Yaskawa INFORM job: X2_8B-21B(90,180).JBI

/JOB
//NAME X2_8B-21B(90,180)
///FOLDERNAME X2
//POS
///NPOS 931,931,931,42,0,0
///TOOL 0
///POSTYPE PULSE
///PULSE
C00000=-1415,-134459,-133802,-1969,12985,79332
C00001=-87080,-112473,-103627,-41798,51237,70410
C00002=-91681,-107347,-99471,-39221,49165,68848
C00003=-93439,-105106,-97054,-38371,48113,68361
C00004=-93441,-104864,-95967,-38672,47682,68565
C00005=-93504,-104969,-96260,-38564,47753,68495
C00006=-95585,-102642,-95415,-36914,47385,67494
C00007=-93504,-104969,-96260,-38564,47753,68495
C00008=-87147,-112175,-102116,-42180,50619,70689
C00009=-87145,-119394,-106475,-25944,48524,38750
C00010=-91166,-110510,-101811,-22693,48895,36705
C00011=-92650,-107060,-99920,-21494,49065,35962
C00012=-94767,-104655,-99060,-19829,49198,34943
C00013=-94484,-105085,-99259,-20052,49173,35080
C00014=-93721,-102513,-96995,-20598,49294,35408
C00015=-94484,-105085,-99259,-20052,49173,35080
C00016=-89209,-117497,-105909,-24366,48468,37757
C00017=-93166,-113214,-115710,-1969,57926,79332
C00018=-93710,-106990,-108704,-1652,56802,79139
C00019=-93766,-106412,-107148,-1629,56140,79127
C00020=-93768,-106433,-106329,-1638,55626,79135
C00021=-93918,-105383,-106173,-1535,56065,79069
C00022=-94164,-101296,-104676,-1361,57240,78956
C00023=-93895,-105502,-106499,-1547,56205,79076
C00024=-93151,-113316,-114305,-1998,57010,79354
C00025=-81072,-99391,-111155,-4750,63110,78553
C00026=-81984,-95120,-104767,-4287,61328,78293
C00027=-82103,-94682,-103397,-4241,60705,78273
C00028=-82106,-94924,-102383,-4271,59960,78300
C00029=-82089,-94934,-102578,-4276,60076,78302
C00030=-82803,-90374,-100753,-3806,61258,77993
C00031=-82089,-94934,-102578,-4276,60076,78302
C00032=-81057,-100006,-109908,-4804,62030,78604
C00033=-94004,-119945,-107122,49530,42714,48164
C00034=-93972,-116281,-97047,53343,39935,45878
C00035=-92833,-103149,-88492,51302,40218,47068
C00036=-93174,-100930,-87132,51219,40604,47120
C00037=-93174,-100493,-85792,51770,40220,46795
C00038=-93174,-101015,-87399,51095,40684,47186
C00039=-92955,-97894,-86230,50180,41136,47726
C00040=-93303,-100448,-87190,51023,40860,47230
C00041=-98055,-98607,-86499,53149,43882,46024
C00042=-96642,-96320,-85623,51883,43475,46780
C00043=-95342,-96864,-85830,51299,42647,47109
C00044=-97130,-98187,-86063,52744,43317,46271
C00045=-114545,-105110,-100746,39625,57097,48369
C00046=-113947,-102413,-97570,39574,56382,48359
C00047=-113947,-102278,-96691,39772,56015,48196
C00048=-113346,-99976,-96570,39024,56612,48763
C00049=-112899,-98120,-95866,38597,56823,49078
C00050=-114020,-99555,-96940,39169,57262,48705
C00051=-56302,-84822,-83054,-58022,66572,84014
C00052=-58361,-85953,-83540,-57558,65172,83717
C00053=-56302,-84822,-83054,-58022,66572,84014
C00054=-50122,-85714,-86741,-59061,71306,84454
C00055=-54195,-101901,-111197,-24063,62262,77343
C00056=-67243,-111926,-101536,21450,29925,69540
C00057=-66442,-101704,-94400,19916,30532,70304
C00058=-66308,-99858,-92576,19846,30336,70336
C00059=-66311,-99589,-91307,20230,29731,70137
C00060=-66308,-99960,-93112,19687,30597,70418
C00061=-70591,-100617,-92786,25268,31264,67678
C00062=-70591,-100325,-91437,25755,30647,67424
C00063=-68222,-99738,-91214,22742,30105,68906
C00064=-70591,-100606,-92729,25289,31242,67667
C00065=-66097,-110297,-96199,21577,27345,69446
C00066=-65719,-107666,-92844,21562,26575,69447
C00067=-65848,-106528,-92445,21497,26927,69482
C00068=-65365,-110699,-93884,21743,25627,69354
C00069=-67243,-111926,-101536,21450,29925,69540
C00070=-68963,-41843,-96211,-398,96948,-48811
C00071=-76932,-51697,-92360,2602,89609,-51106
C00072=-71886,-45093,-85416,705,88639,-49643
C00073=-71886,-45937,-84760,705,87803,-49648
C00074=-71886,-44632,-85753,705,89084,-49641
C00075=-68776,-90352,-95136,-4313,51281,-47645
C00076=-68803,-86754,-93636,-4241,52203,-47695
C00077=-68762,-92243,-95906,-4353,50785,-47617
C00078=-77446,-64871,-91176,8832,74282,-49527
C00079=-75907,-64612,-91046,8095,74185,-49034
C00080=-78150,-64967,-91224,9168,74335,-49752
C00081=-78150,-57569,-97635,8943,81990,-49191
C00082=-68963,-41843,-96211,-398,96948,-48811
C00083=-67385,-42511,-92598,-992,94393,-48367
C00084=-66773,-44328,-90253,-1220,92024,-48175
C00085=-66900,-44765,-89647,-1171,91425,-48205
C00086=-66773,-43962,-90441,-1221,92327,-48178
C00087=-69817,-49291,-93527,-72,91467,-49038
C00088=-102407,-61387,-79216,48101,75803,-74984
C00089=-99741,-62884,-79905,47237,74215,-74494
C00090=-102407,-61387,-79216,48101,75803,-74984
C00091=-71396,-101707,-96198,105,39560,-49678
C00092=-71544,-99303,-95354,247,40276,-49753
C00093=-71126,-105930,-97636,-165,38275,-49535
C00094=-74447,-120283,-111838,3099,39699,-51260
C00095=-57750,-84762,-113304,-22338,79933,-80646
C00096=-38298,-117376,-123136,-35520,84192,-83183
C00097=-31003,-114098,-105660,-45955,85390,-81321
C00098=-32496,-116782,-107403,-45795,84408,-81579
C00099=-34116,-118987,-108120,-45640,83088,-81742
C00100=-33779,-118873,-108083,-45678,83285,-81673
C00101=-33779,-118389,-106291,-45736,82677,-81394
C00102=-33116,-116007,-107005,-45711,84199,-81779
C00103=-43122,-77390,-91933,-43525,86904,-87571
C00104=-44353,-78017,-92219,-43231,86215,-87819
C00105=-45440,-79271,-92786,-42975,85486,-87990
C00106=-45102,-79332,-92813,-43057,85636,-87902
C00107=-45102,-79709,-91490,-43095,84888,-87585
C00108=-41853,-68825,-87871,-43817,88900,-87868
C00109=-48095,-31712,-66541,-47290,99218,-86920
C00110=-48762,-33638,-67810,-47108,98755,-86994
C00111=-49503,-35735,-69173,-46902,98237,-87073
C00112=-49389,-35416,-68966,-46933,98317,-87062
C00113=-49389,-36060,-68028,-46814,97684,-86756
C00114=-48487,-32850,-67294,-47182,98948,-86964
C00115=-45126,-25671,-76382,-49967,106798,-89554
C00116=-48508,-32956,-85951,-38791,109748,-85822
C00117=-73491,-115415,-129730,-12591,84406,-82629
C00118=-68604,-111632,-124361,34026,103601,-55041
C00119=-52690,-105642,-114364,31889,95098,-51390
C00120=-51347,-103959,-112740,31690,94497,-51045
C00121=-51347,-104280,-111882,31650,93903,-51212
C00122=-50963,-109237,-114816,31559,93129,-51281
C00123=-54701,-101748,-112541,32228,96580,-51739
C00124=-54580,-102143,-110625,32107,95358,-52042
C00125=-52710,-105778,-111943,31798,93771,-51772
C00126=-54580,-102143,-110625,32107,95358,-52042
C00127=-53574,-106836,-112314,31893,93817,-52092
C00128=-52008,-102475,-110737,31756,94333,-51344
C00129=-53574,-106836,-112314,31893,93817,-52092
C00130=-61074,-96775,-114868,33501,102293,-52496
C00131=-149084,-102156,-129577,22032,95315,-42360
C00132=-128569,-114069,-129208,14930,94899,-36248
C00133=-124702,-111484,-125119,14131,93099,-35189
C00134=-123206,-111006,-122572,13804,91571,-34868
C00135=-123205,-111346,-122108,13798,91123,-34918
C00136=-123169,-110975,-122344,13795,91444,-34870
C00137=-122647,-104244,-120003,13724,93323,-34489
C00138=-123169,-110975,-122344,13795,91444,-34870
C00139=-116503,-109521,-121739,12400,90787,-32743
C00140=-113941,-110266,-121994,11839,90202,-31960
C00141=-116503,-109521,-121739,12400,90787,-32743
C00142=-121595,-114825,-128025,13496,92670,-34216
C00143=-123984,-121300,-124584,22039,85383,-28695
C00144=-118596,-113071,-118409,20758,84424,-26972
C00145=-117828,-112575,-117002,20585,83663,-26833
C00146=-117596,-112721,-116348,20543,83158,-26838
C00147=-117643,-112201,-116474,20543,83493,-26797
C00148=-117846,-106122,-114344,20549,85245,-26570
C00149=-117643,-112201,-116474,20543,83493,-26797
C00150=-125192,-113488,-115877,22341,84450,-29296
C00151=-124919,-116220,-115928,22323,83104,-29449
C00152=-122352,-116155,-116251,21738,82647,-28614
C00153=-124919,-116220,-115928,22323,83104,-29449
C00154=-123984,-121300,-124584,22039,85383,-28695
C00155=-86442,-134681,-133724,-19248,79211,-32552
C00156=-86002,-121949,-124889,-19319,80358,-32581
C00157=-85994,-121959,-123892,-19351,79775,-32484
C00158=-85995,-122137,-123177,-19379,79272,-32404
C00159=-85938,-122450,-123568,-19392,79360,-32398
C00160=-86651,-115539,-121342,-19081,81262,-32951
C00161=-85938,-122450,-123568,-19392,79360,-32398
C00162=-130270,-119263,-121891,15868,79169,-48216
C00163=-132135,-133974,-122544,16883,72658,-49767
C00164=-129371,-136174,-123179,16117,71390,-48932
C00165=-132135,-133974,-122544,16883,72658,-49767
C00166=-120611,-122953,-119681,21560,80854,-22535
C00167=-120610,-122943,-118608,21593,80243,-22645
C00168=-120610,-122853,-116921,21650,79318,-22813
C00169=-120610,-122881,-117271,21638,79506,-22779
C00170=-120610,-122878,-117279,21638,79511,-22778
C00171=-120610,-122881,-117271,21638,79506,-22779
C00172=-120610,-122873,-117198,21640,79468,-22785
C00173=-120610,-122853,-117190,21640,79473,-22785
C00174=-120610,-122873,-117198,21640,79468,-22785
C00175=-120611,-122910,-120952,21522,81605,-22399
C00176=-120612,-120891,-127143,3106,87300,-4415
C00177=-120611,-122177,-124352,3111,84925,-4474
C00178=-120611,-122645,-122467,3116,83527,-4507
C00179=-120611,-122779,-121606,3119,82929,-4523
C00180=-120611,-122697,-122159,3117,83311,-4513
C00181=-120611,-122692,-122166,3117,83318,-4513
C00182=-120611,-122697,-122159,3117,83311,-4513
C00183=-120611,-121412,-126223,3107,86468,-4436
C00184=-96873,-136971,-131305,19961,95014,-27830
C00185=-53188,-122774,-119059,34227,101931,-42117
C00186=-53187,-122644,-116623,34032,100735,-42492
C00187=-53184,-122447,-115007,33919,99986,-42724
C00188=-53180,-122268,-113886,33849,99484,-42877
C00189=-53186,-122531,-115629,33961,100272,-42636
C00190=-53233,-122033,-113114,32057,113501,-44659
C00191=-53229,-122037,-113108,32057,113495,-44659
C00192=-53233,-122033,-113114,32057,113501,-44659
C00193=-53127,-122157,-112856,34567,84618,-41563
C00194=-53132,-122146,-112848,34568,84621,-41564
C00195=-53127,-122157,-112856,34567,84618,-41563
C00196=-53124,-122720,-116247,34514,86111,-41098
C00197=-68676,-133744,-131015,10578,108811,-68614
C00198=-80160,-118182,-130261,-41,125141,-81817
C00199=-80187,-122370,-123619,-70,118933,-81856
C00200=-80183,-122639,-122398,-68,118043,-81854
C00201=-80181,-122756,-121636,-67,117515,-81853
C00202=-80184,-122603,-122588,-68,118179,-81854
C00203=-80182,-122615,-122584,-67,118170,-81853
C00204=-80184,-122603,-122588,-68,118179,-81854
C00205=-80200,-121154,-126606,-75,121396,-81862
C00206=-109164,-117358,-132635,-7350,119146,-48306
C00207=-144183,-119511,-130571,-15498,107286,-7245
C00208=-197934,-122815,-127402,-28006,89082,55776
C00209=-202772,-123889,-124791,-27048,85608,54814
C00210=-204705,-124106,-122314,-26692,83530,54575
C00211=-204705,-124189,-120905,-26732,82711,54762
C00212=-205113,-122699,-120601,-26621,83104,54520
C00213=-208506,-122040,-120392,-25870,82241,53457
C00214=-204510,-125657,-121990,-26775,82699,54838
C00215=-204510,-125393,-124777,-26704,84359,54459
C00216=-217123,-144581,-130617,-26990,80795,43719
C00217=-208514,-157553,-136215,-22784,79668,13108
C00218=-208514,-151468,-127497,-22936,77598,13510
C00219=-209226,-147410,-126429,-22728,78719,13024
C00220=-208514,-151468,-127497,-22936,77598,13510
C00221=-208514,-156517,-134755,-22805,79329,13174
C00222=-187736,-116553,-120968,-36188,98329,31010
C00223=-144869,-104708,-130913,697,92502,-12445
C00224=-97478,-100538,-119508,25976,122096,-72949
C00225=-94415,-115583,-120723,24602,114867,-73486
C00226=-94145,-116737,-119872,24403,113768,-73630
C00227=-94090,-116915,-118863,24267,113100,-73760
C00228=-94227,-118887,-121662,24392,113788,-73658
C00229=-94618,-126072,-123928,23885,111795,-74261
C00230=-93811,-121058,-122280,24303,112998,-73673
C00231=-123165,-134656,-120887,30393,109989,-65140
C00232=-122877,-135920,-118822,30065,108215,-65520
C00233=-120918,-135771,-118381,30417,107339,-64954
C00234=-122877,-135920,-118822,30065,108215,-65520
C00235=-123434,-129548,-123417,31323,113703,-64157
C00236=-126606,-101457,-128935,16844,101795,-36174
C00237=-152779,-135138,-131563,2515,76140,-19155
C00238=-150820,-122490,-124749,1875,78392,-18455
C00239=-150097,-118368,-121531,1645,78513,-18212
C00240=-150095,-118599,-120646,1648,77850,-18220
C00241=-147666,-112236,-119185,871,80184,-17389
C00242=-146670,-110099,-118456,556,80825,-17059
C00243=-148658,-114325,-119887,1186,79554,-17722
C00244=-87079,-91764,-103818,-42328,107533,9448
C00245=-87027,-91004,-101788,-42122,106912,9740
C00246=-89264,-90509,-101588,-42089,105978,9119
C00247=-87027,-91004,-101788,-42122,106912,9740
C00248=-87391,-90282,-107909,-43186,109836,8282
C00249=-92115,-87061,-118989,-19004,94950,-3823
C00250=-78975,-130870,-123203,19746,71053,-12291
C00251=-74317,-97013,-111518,17407,83606,-9286
C00252=-74211,-95430,-110119,17377,83539,-9259
C00253=-74211,-95892,-109317,17397,82840,-9358
C00254=-75305,-113551,-114600,17838,69768,-10493
C00255=-78326,-111051,-111958,19079,70114,-11550
C00256=-78379,-106110,-110225,18937,71523,-11339
C00257=-78263,-116865,-113913,19272,68408,-11810
C00258=-85880,-113569,-112821,22054,71256,-14152
C00259=-85920,-114580,-110580,22309,69503,-14507
C00260=-82054,-114988,-110714,20879,68380,-13249
C00261=-85920,-114580,-110580,22309,69503,-14507
C00262=-78975,-130870,-123203,19746,67177,-12291
C00263=-159950,-115131,-126913,-23322,109234,64770
C00264=-163413,-124246,-126581,-22686,103792,64589
C00265=-164859,-127477,-125491,-22457,101245,64551
C00266=-164857,-127553,-124648,-22406,100728,64651
C00267=-164862,-127370,-126252,-22506,101730,64457
C00268=-158275,-145382,-129341,-21795,96649,67831
C00269=-159759,-153222,-131425,-21726,93697,67826
C00270=-158275,-145382,-129341,-21795,96649,67831
C00271=-157577,-144643,-126617,-21696,95625,68274
C00272=-160219,-140867,-125578,-21868,96138,67212
C00273=-157577,-144643,-126617,-21696,95625,68274
C00274=-152631,-134238,-128202,-21932,102817,68768
C00275=-146941,-123801,-133763,-3444,102850,52685
C00276=-136178,-116173,-124987,31736,84906,22811
C00277=-134413,-106132,-117362,31242,84680,23412
C00278=-134231,-105594,-115694,31219,83968,23286
C00279=-134230,-105863,-115134,31239,83552,23172
C00280=-134007,-104199,-114803,31151,84035,23389
C00281=-133473,-100630,-113499,30965,84737,23780
C00282=-134315,-106237,-115533,31260,83629,23161
C00283=-136272,-117460,-124003,31807,83855,22481
C00284=-136226,-116324,-125056,31750,84893,22789
C00285=-134474,-106353,-117504,31259,84679,23389
C00286=-134275,-105758,-115681,31235,83904,23252
C00287=-134274,-105987,-115198,31252,83547,23154
C00288=-134027,-104733,-115029,31162,83924,23350
C00289=-133465,-100971,-113658,30966,84667,23763
C00290=-134308,-106598,-115693,31262,83551,23142
C00291=-136269,-117902,-124178,31812,83752,22453
C00292=-139753,-124875,-130430,383,75663,-26245
C00293=-143223,-157944,-133481,-5653,58679,-38405
C00294=-140983,-144085,-126452,-6488,61628,-37698
C00295=-140148,-138933,-122655,-6835,62006,-37402
C00296=-140147,-138616,-121921,-6853,61719,-37384
C00297=-140691,-136506,-121897,-6553,62737,-37651
C00298=-138669,-131542,-120459,-7325,64564,-37004
C00299=-140691,-136506,-121897,-6553,62737,-37651
C00300=-145148,-139028,-124584,-4588,62787,-39337
C00301=-159973,-92454,-110285,14523,90938,-48717
C00302=-158765,-97223,-112137,14224,89465,-48492
C00303=-159973,-92454,-110285,14523,90938,-48717
C00304=-164681,-91509,-114703,15696,94847,-49769
C00305=-142525,-105883,-132766,-7713,103357,-60336
C00306=-90751,-115691,-121566,-36045,104861,-61043
C00307=-92920,-122587,-117773,-35137,99152,-60047
C00308=-93124,-123070,-117553,-35091,98753,-60003
C00309=-93124,-123008,-116878,-35050,98435,-59900
C00310=-93160,-123063,-117190,-35068,98555,-59953
C00311=-95752,-125144,-117838,-34977,96947,-60505
C00312=-93160,-123063,-117190,-35068,98555,-59953
C00313=-92038,-109836,-114685,-38536,89453,-57060
C00314=-86810,-100893,-104585,-47463,92019,-56975
C00315=-88449,-102594,-103600,-47188,90148,-56855
C00316=-88449,-102618,-102426,-47172,89639,-56610
C00317=-88449,-102603,-103366,-47184,90046,-56806
C00318=-85133,-99388,-102162,-47637,92393,-56350
C00319=-85168,-99488,-101153,-47595,91912,-56132
C00320=-86978,-101259,-101820,-47360,90627,-56378
C00321=-84037,-98201,-102123,-47804,93363,-56297
C00322=-108771,-112096,-123986,-16313,85813,-59347
C00323=-109769,-112695,-132242,-3132,99947,-61138
C00324=-127404,-127157,-120795,27540,73197,-60883
C00325=-120526,-123085,-115007,25540,69700,-59025
C00326=-119461,-122312,-114032,25210,69192,-58723
C00327=-119461,-122116,-113003,25293,68708,-58832
C00328=-119461,-122312,-114032,25210,69192,-58723
C00329=-94655,-112249,-115827,-1041,75214,-51009
C00330=-93364,-111129,-115444,-1499,75574,-50577
C00331=-121213,-123445,-114215,25873,69302,-59387
C00332=-127714,-127278,-119628,27738,72603,-61150
C00333=-140848,-129628,-128054,17424,84805,-27418
C00334=-127903,-106251,-120637,17388,91568,-15860
C00335=-124887,-98361,-114445,16717,91208,-14907
C00336=-124614,-94849,-112077,16660,91489,-14780
C00337=-117832,-103976,-115449,15062,87719,-13014
C00338=-118209,-109888,-118953,15141,86934,-13233
C00339=-120968,-118649,-124805,15800,86569,-14208
C00340=-112726,-101228,-128594,1890,90279,15897
C00341=-102865,-105549,-130121,-1361,88970,18873
C00342=-85416,-143080,-122146,-23399,58401,32529
C00343=-89847,-131888,-116792,-20882,59491,30436
C00344=-92125,-126361,-114096,-19602,60042,29398
C00345=-92108,-126361,-114086,-19611,60041,29405
C00346=-94963,-119193,-112807,-13876,65309,25883
C00347=-99230,-109273,-111594,-7832,72910,21884
C00348=-97558,-114678,-114533,-8498,72116,22521
C00349=-94805,-124749,-120489,-9597,70928,23580
C00350=-89899,-115674,-129227,-15589,81503,27304
C00351=-94000,-113154,-130859,1035,116659,-75004
C00352=-93721,-118000,-129934,5060,122177,-74127
C00353=-93715,-120352,-127357,4900,119392,-74256
C00354=-95346,-120435,-125547,4467,118331,-74923
C00355=-87734,-123112,-126247,6115,116903,-72103
C00356=-93725,-120284,-127319,4898,119404,-74259
C00357=-93731,-117931,-129895,5059,122189,-74130
C00358=-92605,-107385,-114202,-42080,118626,-78084
C00359=-94957,-117308,-114744,-40643,113912,-77125
C00360=-96859,-119647,-113709,-40343,111617,-77062
C00361=-96820,-119688,-113698,-40330,111613,-77042
C00362=-92369,-120637,-111842,-39132,112371,-75247
C00363=-87506,-133441,-114197,-38673,106213,-75021
C00364=-90618,-118755,-112828,-39302,114392,-75239
C00365=-88476,-109244,-112462,-40625,118981,-76164
C00366=-73726,-95231,-122050,-23824,117115,-78775
C00367=-68964,-113071,-130294,19412,109419,-80322
C00368=-55630,-112625,-122011,35520,97927,-81697
C00369=-52390,-118820,-120628,34805,93310,-81881
C00370=-47869,-106069,-116317,31727,98681,-78960
C00371=-58944,-112669,-113031,37596,97582,-82877
C00372=-56690,-122472,-119439,35129,92879,-83747
C00373=-59872,-116629,-120975,35716,97415,-83571
C00374=-61517,-148095,-119735,48293,75564,-80066
C00375=-55473,-148057,-116974,48060,71191,-79214
C00376=-53771,-146175,-114985,47935,70110,-78894
C00377=-54494,-144748,-112549,48210,69974,-79344
C00378=-55476,-147094,-115701,48129,70996,-79318
C00379=-61520,-147186,-118480,48348,75358,-80173
C00380=-69196,-132761,-125763,48066,87564,-77891
C00381=-67178,-112107,-133350,-9560,121946,-71499
C00382=-53652,-115588,-130730,-10921,119132,-80041
C00383=-53631,-118653,-128170,-10572,116038,-79726
C00384=-49406,-129162,-130962,-9295,109096,-77614
C00385=-56866,-119557,-126808,-10903,114346,-80761
C00386=-54665,-117852,-125979,-10629,114989,-80007
C00387=-57520,-119011,-127190,-3009,114777,-80027
C00388=-59278,-121853,-127991,842,113579,-80159
C00389=-55695,-120300,-124998,1328,112531,-78914
C00390=-53493,-120154,-126714,1639,113579,-78070
C00391=-53512,-117734,-129516,1682,116546,-78033
C00392=-64263,-112177,-127274,18013,116425,-52133
C00393=-53349,-113292,-116223,34708,105130,-41711
C00394=-53347,-113647,-113946,34435,103813,-42137
C00395=-52680,-112871,-112467,34368,103124,-42082
C00396=-58031,-122280,-112065,36284,98076,-45699
C00397=-53343,-113729,-112902,34324,103242,-42318
C00398=-53345,-113489,-115217,34581,104530,-41905
C00399=-83368,-135406,-127982,43757,111124,24122
C00400=-107112,-148704,-121184,48737,110155,73723
C00401=-107085,-142005,-111593,48000,108472,72828
C00402=-107084,-140010,-108705,47787,107957,72557
C00403=-87331,-137626,-115833,38185,104318,80918
C00404=-107143,-152743,-127540,-1092,113262,57657
C00405=-96955,-158208,-128899,-2670,111185,56030
C00406=-107130,-144670,-115956,-40497,90070,47196
C00407=-107133,-145289,-116877,-40503,90261,47122
C00408=-107139,-146938,-119316,-40521,90762,46927
C00409=-81304,-146505,-131302,-46256,99624,33732
C00410=-42290,-135810,-134986,-6789,56953,-43412
C00411=-53482,-111499,-99357,-5283,31563,-44884
C00412=-53488,-110753,-96932,-5448,30458,-44798
C00413=-53106,-110845,-96482,-5998,30161,-44520
C00414=-53143,-110117,-93832,-6189,28906,-44421
C00415=-53188,-109818,-93168,-6175,28651,-44427
C00416=-53095,-108922,-90553,-6542,27518,-44240
C00417=-53472,-108968,-91791,-5862,28222,-44586
C00418=-53466,-109889,-94290,-5675,29282,-44681
C00419=-93748,-113667,-111432,27227,62688,-41579
C00420=-93751,-113561,-109328,27520,61581,-41869
C00421=-94535,-110348,-107800,27711,62471,-41963
C00422=-94560,-109570,-102150,28499,59749,-42715
C00423=-93743,-112935,-104615,28181,59286,-42489
C00424=-93741,-113330,-106821,27872,60309,-42206
C00425=-53707,-103235,-126817,-3349,90409,-72793
C00426=-53694,-107630,-124107,-3352,86490,-72685
C00427=-53689,-108955,-122884,-3357,85060,-72645
C00428=-53697,-108940,-122873,-3354,85062,-72648
C00429=-53721,-108898,-122839,-3346,85062,-72656
C00430=-53729,-108884,-122827,-3345,85059,-72658
C00431=-53735,-107561,-124050,-3339,86489,-72698
C00432=-53748,-103173,-126762,-3336,90406,-72805
C00433=-44251,-68518,-112793,-6305,100072,-70363
C00434=-80270,30794,-42629,-11133,115571,-76543
C00435=-69737,67118,16632,-42575,112328,-80617
C00436=-69636,63823,22197,-49512,110599,-81416
C00437=-67564,55530,12856,-50142,112647,-81508
C00438=-66424,44944,1253,-49852,108764,-84350
C00439=-65618,29495,-14632,-48008,102670,-88237
C00440=-64581,15750,-27557,-48396,103780,-88326
C00441=-64160,11595,-31362,-48525,104124,-88308
C00442=-61878,-10748,-50140,-48981,105285,-87846
C00443=-62672,195,-41330,-51307,112408,-84907
C00444=-58944,10301,-35991,-52571,115494,-84879
C00445=-69716,-6230,-69222,-29298,97742,-75748
C00446=-102330,-22799,-82036,11222,88832,-73278
C00447=-48313,-118911,-129560,19207,92704,-27073
C00448=-53495,-110604,-121584,20154,93282,-28749
C00449=-53898,-112894,-120750,20179,91787,-29140
C00450=-54091,-109968,-119805,20238,92698,-29053
C00451=-54227,-109896,-119946,20266,92849,-29073
C00452=-54259,-112639,-122766,20278,93161,-29031
C00453=-53522,-108468,-123882,20258,95652,-28360
C00454=-66910,-101677,-117691,1645,82254,17515
C00455=-66905,-103395,-115374,1652,79946,17486
C00456=-66559,-103374,-114061,1536,79140,17588
C00457=-66525,-103141,-114029,1523,79241,17602
C00458=-67620,-103650,-114144,1902,79074,17240
C00459=-69811,-106122,-108316,12679,69437,17327
C00460=-66783,-105788,-110032,11324,70201,18483
C00461=-66785,-105108,-112553,11207,72068,18659
C00462=-34610,-119076,-126707,-31995,89279,47352
C00463=-26693,-119602,-105841,-51320,82883,62074
C00464=-26676,-118953,-103885,-51392,82336,62389
C00465=-26611,-118260,-103653,-51381,82509,62328
C00466=-26639,-116853,-99731,-51529,81413,62927
C00467=-26666,-118021,-101324,-51491,81640,62785
C00468=-26683,-118745,-103309,-51412,82173,62476
C00469=-26741,-121947,-116429,-51038,86269,60171
C00470=-80158,-111738,-121779,-46707,81282,-33331
C00471=-80124,-114295,-114082,-47454,77096,-31277
C00472=-80115,-114367,-110881,-47781,75720,-30584
C00473=-79927,-114969,-109893,-47987,75192,-30221
C00474=-79885,-115119,-109957,-48003,75187,-30197
C00475=-80052,-114603,-110983,-47806,75713,-30548
C00476=-80061,-114542,-114188,-47480,77086,-31241
C00477=-80063,-113108,-120040,-30435,104055,-77976
C00478=-80050,-114212,-116860,-30086,101864,-77373
C00479=-80380,-112077,-114717,-30053,101557,-77419
C00480=-79932,-114590,-112006,-35005,85347,-77215
C00481=-79912,-114566,-112044,-35008,85386,-77219
C00482=-80479,-112475,-109427,-36632,80098,-77307
C00483=-80029,-114714,-111597,-36713,80437,-77233
C00484=-82440,-93132,-104306,-35744,84828,-79668
C00485=-83378,-90315,-100640,-35536,83784,-79702
C00486=-86724,-76310,-94495,-34501,85296,-81493
C00487=-81341,-82881,-101909,-35963,88366,-80388
C00488=-80042,-114535,-115070,-36542,82240,-77847
C00489=-80040,-111621,-122742,-8414,85267,-41918
C00490=-80035,-113457,-119567,-8450,82400,-41723
C00491=-81798,-124774,-120168,-7328,73182,-41674
C00492=-80327,-109577,-118133,2572,87034,-53415
C00493=-79380,-112621,-119090,2349,86031,-53125
C00494=-78889,-114029,-118891,6085,83597,-58153
C00495=-80002,-113603,-119620,10752,83390,-63441
C00496=-80006,-103113,-128729,10775,94202,-62513
C00497=-39776,-103787,-110683,-21075,62663,59255
C00498=-39766,-104399,-107995,-21452,60825,59622
C00499=-41663,-99518,-106576,-17765,63773,58656
C00500=-39441,-104963,-106701,-21848,59898,59942
C00501=-39326,-105104,-106740,-21922,59881,59993
C00502=-39744,-104425,-108009,-21464,60826,59630
C00503=-39754,-103814,-110697,-21087,62664,59263
C00504=-47977,-106691,-119962,-23629,83327,62671
C00505=-66867,-99660,-121232,-22132,99220,62132
C00506=-66851,-102572,-118810,-21937,96446,62653
C00507=-74494,-137000,-128982,-14609,78071,53501
C00508=-72467,-138184,-128020,-15181,77278,54315
C00509=-67516,-140688,-126942,-16493,76361,56201
C00510=-43056,-127353,-114280,-36292,85121,62743
C00511=-66851,-103895,-117201,-21852,94891,62938
C00512=-66868,-101493,-119792,-22004,97521,62449
C00513=-74321,-107832,-126985,11736,80239,61811
C00514=-66584,-114412,-108983,34198,49386,64476
C00515=-66581,-113854,-105403,35147,47795,63826
C00516=-59001,-125725,-103773,32485,32454,61113
C00517=-65790,-113886,-101008,36132,45231,63145
C00518=-65568,-123466,-98279,45853,34675,56822
C00519=-65581,-123771,-97752,46366,34344,56544
C00520=-66567,-113311,-102857,35821,46729,63375
C00521=-66569,-114089,-106515,34851,48256,64025
C00522=-66614,-114312,-115902,32344,53032,65825
C00523=-26293,-124733,-123676,35115,86081,77095
C00524=-26278,-124914,-120130,35186,84196,76502
C00525=-26550,-125631,-118910,35285,83385,76132
C00526=-26140,-123752,-118256,35186,83681,76394
C00527=-26301,-124893,-120124,35190,84211,76498
C00528=-26317,-124710,-123669,35119,86096,77090
C00529=-26368,-124828,-121889,39154,95960,78120
C00530=-26350,-124746,-118556,38992,94373,77544
C00531=-26342,-124553,-116950,38932,93670,77290
C00532=-26340,-123995,-113991,38847,92461,76851
C00533=-26347,-124286,-115407,38884,93032,77056
C00534=-26365,-124761,-118865,39006,94524,77592
C00535=-26264,-124528,-116402,47920,86072,68134
C00536=-26249,-123768,-112787,47988,84810,67516
C00537=-26243,-123374,-111311,48022,84325,67278
C00538=-26226,-122772,-109280,48074,83674,66962
C00539=-26232,-123227,-110778,48035,84146,67194
C00540=-26247,-124165,-114452,47952,85370,67795
C00541=-82585,-123093,-118421,52491,64599,59558
C00542=-107155,-118824,-102398,58122,50036,52281
C00543=-107155,-117467,-98958,59145,49269,51564
C00544=-96813,-117817,-104188,42223,47347,50994
C00545=-105933,-121077,-109912,10415,42869,62990
C00546=-105953,-121074,-109843,10442,42831,62975
C00547=-107149,-121400,-109798,11502,42801,62375
C00548=-106717,-121349,-105974,7567,38238,71665
C00549=-107169,-120346,-107141,7797,39493,71540
C00550=-108433,-119625,-117514,7930,46308,71537
C00551=-107111,-122100,-111275,39348,45202,56077
C00552=-107109,-117760,-98763,43179,41028,53713
C00553=-106761,-117495,-97713,43363,40478,53604
C00554=-106458,-119074,-102370,12274,36991,61895
C00555=-94483,-118196,-102129,-13006,37418,75653
C00556=-107097,-114092,-90505,-56996,42891,80282
C00557=-107127,-114270,-91297,-56630,43098,80056
C00558=-101354,-119078,-102486,-55464,49091,79315
C00559=-93612,-109275,-133010,12113,75674,64968
C00560=-74458,-81913,-116300,25886,107898,47202
C00561=-74285,-84923,-113224,25351,104735,46539
C00562=-74085,-86300,-112083,25142,103399,46313
C00563=-71499,-76504,-108067,25490,106819,45523
C00564=-62961,-60085,-100217,24652,107848,48688
C00565=-60437,-59805,-99888,23461,105440,51393
C00566=-60588,-58283,-100875,23679,106756,51616
C00567=-60637,-54628,-103477,24231,109960,52288
C00568=-76657,-70403,-83915,51355,64349,40407
C00569=-74830,-68241,-74355,53953,55282,38932
C00570=-73110,-62379,-68708,53436,54020,39148
C00571=-73126,-62440,-68450,53549,53912,39057
C00572=-36930,-67607,-75173,-26029,44061,77403
C00573=-80523,-89058,-85253,18218,36719,55154
C00574=-82272,-90569,-85112,18702,34759,56728
C00575=-81508,-95500,-88175,18158,33969,56993
C00576=-81043,-103588,-94156,17854,33413,57140
C00577=-82846,-88179,-88219,41798,48730,43563
C00578=-81818,-81213,-82326,41198,48211,43888
C00579=-79663,-80074,-80946,37957,46333,45127
C00580=-64011,-84834,-85332,4259,39755,58703
C00581=-75846,-87347,-86370,15921,40584,52659
C00582=-47572,-67654,-78731,-37306,60592,66422
C00583=-46339,-68382,-80235,-37741,61555,66618
C00584=-42699,-70655,-83815,-39176,63943,67342
C00585=-43803,-67144,-92021,-36183,69839,64523
C00586=-86906,-70734,-117845,25978,101850,24881
C00587=-194376,-118372,-116958,36622,58194,-75254
C00588=-187943,-106127,-101715,33777,52366,-74665
C00589=-187951,-105693,-98645,34509,50978,-75202
C00590=-187954,-105458,-97394,34809,50440,-75417
C00591=-187960,-105469,-97402,34805,50444,-75420
C00592=-187927,-105629,-98482,19599,46235,-60273
C00593=-187923,-105820,-99644,19403,46817,-60144
C00594=-187914,-106157,-102495,18928,48312,-59826
C00595=-188021,-109107,-91072,54887,40419,-77132
C00596=-188025,-108188,-88773,55807,39869,-77674
C00597=-188027,-107805,-87846,56180,39654,-77892
C00598=-188036,-107761,-87717,56242,39627,-77928
C00599=-188035,-108145,-88644,55869,39841,-77710
C00600=-188030,-109068,-90945,54948,40390,-77168
C00601=-188015,-114130,-110744,41340,72657,-75143
C00602=-188018,-113864,-107763,41683,71368,-75679
C00603=-188019,-113684,-106544,41824,70871,-75888
C00604=-188009,-113674,-106577,41816,70886,-75877
C00605=-188008,-113852,-107795,41674,71383,-75668
C00606=-188005,-114114,-110775,41332,72673,-75132
C00607=-187933,-113872,-110928,18210,58720,-57176
C00608=-187882,-113256,-105308,-719,43762,-42538
C00609=-187896,-112711,-102669,-725,42418,-42533
C00610=-187852,-113170,-101841,-775,41671,-42505
C00611=-187778,-112374,-98354,-1639,37547,-42296
C00612=-187899,-111729,-99017,-1491,38283,-42378
C00613=-187886,-112431,-101600,-1465,39511,-42393
C00614=-192869,-127835,-120494,22551,66263,-53872
C00615=-188079,-122619,-114609,40714,83609,-61664
C00616=-188077,-122103,-112045,40794,82601,-62056
C00617=-188097,-121812,-110726,41966,87288,-59780
C00618=-188097,-121769,-110559,41966,87227,-59806
C00619=-188105,-121282,-108770,41980,86589,-60067
C00620=-188106,-121566,-109755,41972,86936,-59927
C00621=-188110,-122188,-112187,41960,87826,-59570
C00622=-188058,-121965,-125191,40549,88870,-59628
C00623=-104402,-90439,-123637,22599,88102,26907
C00624=-80407,-121901,-119741,18448,66455,46046
C00625=-80400,-121844,-116068,18757,64334,45697
C00626=-80358,-121826,-114599,18875,63477,45568
C00627=-79500,-120626,-114191,18436,63629,45929
C00628=-80475,-121542,-115946,18779,64427,45684
C00629=-80482,-121578,-119613,18469,66554,46034
C00630=-85156,-144709,-129107,-21632,59402,64028
C00631=-93856,-120445,-109825,-39450,57641,70752
C00632=-93847,-119691,-106928,-40019,56559,71233
C00633=-86628,-99816,-98593,-45940,69277,74290
C00634=-86043,-99167,-98859,-45014,69635,74495
C00635=-83318,-93529,-94650,-47165,68336,75996
C00636=-93680,-116508,-100417,-40719,46210,72415
C00637=-93820,-118277,-102341,-40471,46353,72255
C00638=-93828,-119232,-105178,-39715,47322,71755
C00639=-93822,-120125,-107980,-28359,52237,38282
C00640=-93816,-119582,-106091,-28689,51458,38525
C00641=-93813,-119346,-105328,-28822,51152,38622
C00642=-93805,-118409,-102529,-29499,49391,39302
C00643=-93820,-119862,-107056,-29266,59584,40856
C00644=-93823,-120114,-107958,-29147,59957,40747
C00645=-93830,-120670,-110185,-28854,60909,40473
C00646=-63807,-119595,-131717,-32346,77391,31957
C00647=-66677,-122882,-119460,-9954,65715,-31882
C00648=-66675,-122709,-116301,-10101,63887,-31721
C00649=-66675,-122586,-115330,-10147,63360,-31673
C00650=-66678,-122782,-121307,9429,81851,-37654
C00651=-66765,-122962,-121469,9451,81867,-37681
C00652=-66675,-122328,-113778,33290,107246,-42961
C00653=-66675,-122499,-114776,33395,107690,-42822
C00654=-66677,-122795,-117228,33681,108831,-42458
C00655=-66720,-122114,-124411,34847,112827,-41144
C00656=-15972,-110889,-128286,-10965,59905,-43045
C00657=-15972,-110889,-128286,-10965,59905,-43045
C00658=-101389,-60822,-75148,6919,68546,-70102
C00659=-115790,69230,64798,-8053,66131,-71909
C00660=-120688,105020,73307,-12402,84846,-73777
C00661=-120868,103639,75593,-12409,82749,-73629
C00662=-120940,103216,76680,-12418,81872,-73566
C00663=-120940,103732,79019,-12450,80724,-73451
C00664=-120940,103216,76680,-12418,81872,-73566
C00665=-120298,112004,89967,-12640,78393,-72988
C00666=-120707,106255,82361,-12511,80017,-73298
C00667=-120298,112004,89967,-12640,78393,-72988
C00668=-120298,111380,88066,-12608,79223,-73073
C00669=-122096,108036,83635,-12280,79933,-73777
C00670=-122096,108524,85355,-12307,79144,-73698
C00671=-121742,108481,85298,-12365,79210,-73582
C00672=-121911,108228,84384,-12322,79608,-73681
C00673=-120228,112105,88453,-12614,79365,-73063
C00674=-120053,112844,85327,-12571,81642,-73235
C00675=-120830,71540,61874,-4756,55589,-66514
C00676=-120535,76858,72419,-5134,51864,-66212
C00677=-120418,79487,77321,-5314,50212,-66075
C00678=-120418,81305,81326,-5435,48689,-65991
C00679=-120418,79487,77321,-5314,50212,-66075
C00680=-121101,73566,71896,-4942,50464,-66384
C00681=-120640,77942,77238,-5256,49458,-66131
C00682=-121101,73566,71896,-4942,50464,-66384
C00683=-121222,71175,67349,-4775,52021,-66512
C00684=-121527,66226,57370,-4418,55590,-66797
C00685=-120817,46858,51705,6808,46216,-80289
C00686=-120487,52530,62238,7041,42645,-80409
C00687=-120357,55197,66992,7170,41090,-80474
C00688=-120357,57219,71131,7393,39594,-80606
C00689=-120357,55197,66992,7170,41090,-80474
C00690=-121171,51687,64922,7778,40638,-80922
C00691=-120657,55397,69123,7546,39918,-80729
C00692=-121171,51687,64922,7778,40638,-80922
C00693=-121307,49062,60252,7635,42163,-80850
C00694=-121648,43436,49847,7373,45678,-80715
C00695=-109578,66950,51259,-9202,73878,-70224
C00696=-101389,-60822,-75148,6919,68546,-70102
C00697=-96929,-90691,-89138,5080,61517,-23019
C00698=-96929,-90691,-89138,5080,61517,27168
C00699=-133997,38575,-5386,4879,105902,64390
C00700=-134430,35731,-4221,4855,103756,64161
C00701=-134605,34666,-3678,4847,102887,64068
C00702=-134604,34193,-2477,4825,101908,64030
C00703=-134605,34666,-3678,4847,102887,64068
C00704=-133324,38381,1851,4717,101326,64430
C00705=-133984,36157,-436,4773,101627,64224
C00706=-133324,38381,1851,4717,101326,64430
C00707=-132740,42105,45,4739,104308,64739
C00708=-159526,23962,790,32225,80504,55500
C00709=-158922,24925,5721,32299,78113,55050
C00710=-158682,25453,8443,32390,76826,54772
C00711=-158681,25549,9587,32465,76269,54609
C00712=-158682,25408,7790,32348,77149,54866
C00713=-160104,22984,7189,32780,76948,54233
C00714=-159169,24509,8648,32575,76492,54477
C00715=-160104,22984,7189,32780,76948,54233
C00716=-160967,21427,101,32642,80299,54873
C00717=-147551,27169,-6215,28445,81493,60312
C00718=-147017,27605,-1759,28452,79091,59917
C00719=-146805,27803,661,28506,77793,59674
C00720=-146803,27699,1600,28565,77235,59535
C00721=-146805,27874,109,28472,78126,59757
C00722=-148390,24338,-1607,29025,77984,59121
C00723=-147556,26192,183,28786,77573,59333
C00724=-148390,24338,-1607,29025,77984,59121
C00725=-149162,23542,-7999,28991,81344,59682
C00726=-129846,-17397,-52274,16165,101048,68229
C00727=-103949,-6271,-30701,7884,96105,76175
C00728=-94102,16895,-5866,4380,94047,79161
C00729=-94024,14878,-3719,4358,91692,79105
C00730=-93993,14152,-2780,4351,90742,79083
C00731=-93993,14253,-1030,4349,89719,79047
C00732=-93993,14152,-2780,4351,90742,79083
C00733=-93685,20015,4382,4321,89334,79138
C00734=-93881,17120,1686,4338,89515,79078
C00735=-93685,20015,4382,4321,89334,79138
C00736=-93796,22544,1176,4343,92603,79213
C00737=-95224,-25687,-42365,27028,60157,72238
C00738=-94111,-23276,-36997,26973,57954,72128
C00739=-93676,-22245,-34794,26967,57075,72081
C00740=-93677,-22196,-33100,27266,56165,71832
C00741=-93676,-22245,-34794,26967,57075,72081
C00742=-94165,-26445,-35973,27662,55954,71554
C00743=-93910,-23559,-33944,27450,56079,71704
C00744=-94165,-26445,-35973,27662,55954,71554
C00745=-95768,-30118,-43626,27714,58991,71694
C00746=-97625,-41604,-59467,17173,89706,-8843
C00747=-96114,-37688,-53918,16886,88057,-8555
C00748=-95526,-36022,-51615,16777,87400,-8443
C00749=-95527,-36150,-50037,16784,86406,-8579
C00750=-95526,-36022,-51615,16777,87400,-8443
C00751=-95532,-36183,-50637,16782,86745,-8534
C00752=-95234,-33170,-48668,16723,87008,-8396
C00753=-95532,-36183,-50637,16782,86745,-8534
C00754=-95504,-36095,-50208,16778,86530,-8554
C00755=-93996,-36675,-50581,16493,86163,-8084
C00756=-95504,-36095,-50208,16778,86530,-8554
C00757=-97625,-41604,-59467,17173,89706,-8843
C00758=-101873,-77751,-87156,42969,63075,62474
C00759=-95937,-74809,-81328,40948,58735,63434
C00760=-95565,-74583,-80935,40815,58468,63500
C00761=-95566,-74620,-79294,41227,57681,63141
C00762=-95565,-74583,-80935,40815,58468,63500
C00763=-98755,-73227,-80296,42221,60183,62682
C00764=-98803,-73638,-78797,42678,59356,62269
C00765=-96868,-74481,-79195,41849,58298,62761
C00766=-98803,-73638,-78797,42678,59356,62269
C00767=-97163,-69666,-76891,41573,59236,63045
C00768=-96752,-66139,-75134,41097,59602,63417
C00769=-97163,-69666,-76891,41573,59236,63045
C00770=-101873,-77751,-87156,42969,63075,62474
C00771=-126113,-49786,-51573,51544,90004,55144
C00772=-123973,-50127,-48217,51392,87374,54806
C00773=-123286,-49758,-46380,51349,86473,54664
C00774=-118478,-34750,-37348,50925,85086,56432
C00775=-119272,-35479,-39244,50973,86038,56539
C00776=-121232,-35158,-42579,51146,88553,56901
C00777=-111145,-57425,-62081,41633,61582,55088
C00778=-109620,-53993,-56645,41578,59663,54986
C00779=-109014,-52418,-54338,41560,58914,54950
C00780=-105531,-54881,-55720,40219,56972,55856
C00781=-106107,-56401,-57979,40230,57706,55889
C00782=-107578,-60042,-63488,40293,59558,55964
C00783=-93331,-25535,-46307,22677,87971,72102
C00784=-84242,-5399,-27465,11713,100257,81196
C00785=-83743,-8192,-25851,11599,97806,81134
C00786=-83603,-8644,-24372,11558,96668,81075
C00787=-80847,-8673,-24279,11462,96208,81977
C00788=-80973,-8366,-25985,11504,97411,82047
C00789=-81511,-5615,-27635,11617,99868,82095
C00790=-103949,-6271,-30701,7884,96105,76175
C00791=-129846,-17397,-52274,16165,101048,68229
C00792=-175693,57260,35469,48998,74273,48315
C00793=-174652,59964,42108,49342,71909,47593
C00794=-173987,58917,42535,48748,68669,47097
C00795=-173562,58305,42809,47399,62634,46211
C00796=-173482,53917,36869,46602,62532,46609
C00797=-174364,49990,29079,45939,64941,47387
C00798=-163099,39792,11105,47007,80916,54866
C00799=-161954,40669,15666,46993,78691,54338
C00800=-161675,41954,18470,47071,77805,54042
C00801=-160520,35916,12218,46685,77730,54566
C00802=-160850,34862,9687,46632,78611,54832
C00803=-162019,34035,5199,46665,80839,55343
C00804=-147988,42797,109,12455,106225,61454
C00805=-148219,40121,1423,12320,104123,61157
C00806=-146030,57026,21700,8846,110028,61895
C00807=-145258,50191,13883,9166,109401,62129
C00808=-144531,51862,16039,8885,111237,62498
C00809=-146794,35355,-3496,12271,104485,61677
C00810=-146567,38090,-4821,12411,106625,61976
C00811=-96929,-90691,-89138,5080,61517,27168
C00812=-96929,-90691,-89138,5080,61517,-23019
C00813=-101389,-60822,-75148,6919,68546,-70102
C00814=-109578,66950,51259,-9202,73878,-70224
C00815=-119285,73548,61078,-7759,54489,-67872
C00816=-119140,78931,71700,-8230,50768,-67516
C00817=-119018,68322,64494,-9513,43413,-66753
C00818=-123077,79861,78861,-6886,39527,-68452
C00819=-122308,90513,86215,-6785,47517,-68668
C00820=-122473,83260,72935,-6271,51921,-69036
C00821=-119074,82203,59752,-14757,75142,-72556
C00822=-112473,77653,55392,-16315,76732,-70397
C00823=-111583,66581,50085,-22599,68947,-68307
C00824=-112205,67748,51306,-22435,68636,-68485
C00825=-112809,96137,83372,-20713,72479,-69433
C00826=-121067,113951,104217,-8230,68834,-71393
C00827=-120880,99674,85606,-8530,71491,-71499
C00828=-121360,95237,80258,-8447,70766,-71619
C00829=-121396,72779,51526,-8459,68942,-71502
C00830=-134157,70152,49704,15847,72235,-43808
C00831=-133722,73949,59265,16087,68355,-44178
C00832=-133862,75249,62165,16247,67307,-44381
C00833=-129675,65866,51066,4701,64817,-31992
C00834=-128682,62362,47014,4314,65455,-31601
C00835=-130205,57581,36634,4742,69462,-32000
C00836=-130312,54578,33992,4779,69550,-32035
C00837=-129992,46081,35923,20239,67004,8502
C00838=-121496,43425,36833,5893,59088,22773
C00839=-120237,47252,43120,2387,56768,25932
C00840=-119972,47626,45454,2298,55515,26011
C00841=-128073,50557,47782,20949,62737,7811
C00842=-127834,53853,52717,21124,61417,7650
C00843=-123180,48310,46556,9691,56439,19302
C00844=-122651,35401,27095,8965,61652,19959
C00845=-109578,66950,51259,-9202,73878,-70224
C00846=-101389,-60822,-75148,6919,68546,-70102
C00847=-96929,-90691,-89138,5080,61517,-23019
C00848=-93242,-109726,-96296,3420,55961,28393
C00849=-92156,-22649,-39625,10516,94476,60392
C00850=-92549,-23820,-36378,10508,91967,60047
C00851=-92689,-24290,-35079,10509,90961,59915
C00852=-95254,-23373,-34430,10727,91365,59075
C00853=-94898,-22950,-35761,10710,92338,59280
C00854=-94492,-21797,-39017,10723,94837,59633
C00855=-92575,-26977,-42679,21088,73618,56030
C00856=-92430,-25186,-37423,21282,71416,55682
C00857=-92290,-24713,-35488,21345,70493,55566
C00858=-95616,-23226,-34216,23502,71566,54461
C00859=-95477,-23933,-36320,23344,72386,54682
C00860=-95719,-25683,-41558,23174,74597,55037
C00861=-96929,-90691,-89138,5080,61517,27168
C00862=-96929,-90691,-89138,5080,61517,-23019
C00863=-101389,-60822,-75148,6919,68546,-70102
C00864=-109578,66950,51259,-9202,73878,-70224
C00865=-108278,48890,46404,-6655,48460,-73563
C00866=-108252,54023,56228,-7048,45078,-73302
C00867=-107661,40825,52409,-14308,28668,-70428
C00868=-112610,50539,61242,-7713,29705,-74042
C00869=-112702,61866,65174,-4315,43297,-75310
C00870=-112766,56024,54314,-4011,46966,-75508
C00871=-103921,32533,46603,10708,30188,-75698
C00872=-104692,35200,60863,30413,16065,-83251
C00873=-104796,38679,66061,33302,14894,-84599
C00874=-102333,36267,63497,27606,14351,-81669
C00875=-100412,37194,55383,7603,26828,-73795
C00876=-100998,29868,43914,7479,30147,-73786
C00877=-109578,66950,51259,-9202,73878,-70224
C00878=-101389,-60822,-75148,6919,68546,-70102
C00879=-96929,-90691,-89138,5080,61517,-23019
C00880=-96929,-90691,-89138,5080,61517,27168
C00881=-90570,-23240,-39845,-1682,91658,61068
C00882=-90349,-1837,-19216,-4288,101242,62233
C00883=-91120,2554,-13785,-2797,103692,62024
C00884=-91367,5226,-10916,-6319,104184,61643
C00885=-95291,-22836,-35623,-1093,89189,59526
C00886=-94239,-22001,-38963,-1226,91687,59852
C00887=-90424,-29050,-43505,3763,58999,61302
C00888=-86008,-21130,-36360,-6353,62529,61992
C00889=-86454,-19207,-33152,-6175,61515,61881
C00890=-89453,-18520,-32647,-4592,61359,60761
C00891=-95351,-24457,-36663,6763,57473,59317
C00892=-94707,-27619,-42528,6252,59394,59681
C00893=-109011,-26713,-50438,8452,98222,74634
C00894=-144543,31549,-11380,-159,92982,60584
C00895=-143093,45679,4448,-4866,97184,60249
C00896=-142229,53785,16152,-6705,99618,60162
C00897=-144891,70831,35748,-7385,98802,59208
C00898=-148937,42537,3991,922,89189,59187
C00899=-148250,43318,770,754,91565,59420
C00900=-172279,3947,-14828,46151,77384,48319
C00901=-167570,-10636,-17777,41693,62852,42800
C00902=-166655,-7092,-11488,42082,60867,42363
C00903=-169056,5005,-1455,42887,62060,41693
C00904=-172859,17944,7820,47479,72977,45875
C00905=-174013,15583,1984,47261,75226,46421
C00906=-109011,-26713,-50438,8452,98222,74634
C00907=-99312,-50897,-61026,22837,72179,74454
C00908=-98138,-49989,-56545,22703,69739,74412
C00909=-106382,-52347,-50887,37007,65807,70627
C00910=-98813,-18962,-39289,22939,92751,75811
C00911=-101547,-27333,-44313,25543,91651,74875
C00912=-97857,-18198,-39852,20610,99055,76884
C00913=-96922,-25876,-47272,18742,95048,76352
C00914=-97638,-23312,-49453,18962,97729,76524
C00915=-81141,-50558,-66105,12803,46081,75388
C00916=-80687,-46119,-60183,12697,44679,75401
C00917=-80513,-44339,-57785,12667,44105,75401
C00918=-80516,-44488,-54802,13120,42239,75121
C00919=-80690,-46329,-57233,13145,42803,75122
C00920=-81145,-50923,-63237,13239,44177,75109
C00921=-83601,15534,-39616,9664,96262,77072
C00922=-80484,90945,50155,4324,118905,78550
C00923=-80490,84570,45509,4303,118490,78531
C00924=-80493,82108,43801,4293,118276,78521
C00925=-80495,81630,46278,4216,116511,78452
C00926=-80492,84058,47940,4226,116735,78462
C00927=-83493,53381,-2692,9637,111099,78940
C00928=-91945,-14209,-43630,9790,83010,75128
C00929=-10907,-117335,-90652,-18762,63715,-59495
C00930=-15972,-110889,-128286,-10965,59905,-43045
BC00000=48829,688840,1075175
BC00001=366911,902233,1075175
BC00002=366911,902233,1075175
BC00003=366911,902233,1075175
BC00004=366911,902233,1075175
BC00005=366911,902233,1075175
BC00006=366911,902233,1075175
BC00007=366911,902233,1075175
BC00008=366911,902233,1075175
BC00009=333056,895412,1075175
BC00010=333056,895412,1075175
BC00011=333056,895412,1075175
BC00012=333056,895412,1075175
BC00013=333056,895412,1075175
BC00014=333056,895412,1075175
BC00015=333056,895412,1075175
BC00016=333056,895412,1075175
BC00017=358091,902222,1075175
BC00018=358091,902222,1075175
BC00019=358091,902222,1075175
BC00020=358091,902222,1075175
BC00021=358091,902222,1075175
BC00022=358091,902222,1075175
BC00023=358091,902222,1075175
BC00024=358091,902222,1075175
BC00025=398174,894103,1075175
BC00026=398174,894103,1075175
BC00027=398174,894103,1075175
BC00028=398174,894103,1075175
BC00029=398174,894103,1075175
BC00030=398174,894103,1075175
BC00031=398174,894103,1075175
BC00032=398174,894103,1075175
BC00033=264903,781270,1075175
BC00034=264903,781270,1075175
BC00035=264904,781269,1075172
BC00036=264904,781269,1075171
BC00037=264904,781269,1075171
BC00038=264904,781269,1075168
BC00039=264904,781269,1075168
BC00040=264904,781269,1075168
BC00041=264904,781269,1075168
BC00042=264904,781269,1075168
BC00043=264904,781269,1075164
BC00044=264903,781270,1075175
BC00045=301264,775814,1075175
BC00046=301264,775814,1075175
BC00047=301264,775814,1075175
BC00048=301264,775814,1075175
BC00049=301264,775814,1075175
BC00050=301264,775814,1075175
BC00051=301264,775814,1075175
BC00052=301264,775814,1075175
BC00053=301264,775814,1075175
BC00054=301264,775814,1075175
BC00055=274235,786209,1075175
BC00056=238672,799885,1075175
BC00057=238672,799885,1075175
BC00058=238672,799885,1075175
BC00059=238672,799885,1075175
BC00060=238672,799885,1075175
BC00061=238672,799885,1075175
BC00062=238672,799885,1075175
BC00063=238672,799885,1075175
BC00064=238672,799884,1075171
BC00065=238672,799884,1075171
BC00066=238672,799885,1075175
BC00067=238672,799885,1075175
BC00068=238672,799885,1075175
BC00069=238672,799885,1075175
BC00070=318263,750454,1075175
BC00071=318263,750454,1075175
BC00072=318263,750454,1075175
BC00073=318263,750454,1075175
BC00074=318263,750454,1075175
BC00075=318263,750454,1075175
BC00076=318263,750454,1075175
BC00077=318263,750454,1075175
BC00078=318263,750454,1075175
BC00079=318263,750454,1075175
BC00080=318263,750454,1075175
BC00081=318263,750454,1075175
BC00082=318263,750454,1075175
BC00083=318263,750454,1075175
BC00084=318263,750454,1075175
BC00085=318263,750454,1075175
BC00086=318263,750454,1075175
BC00087=318263,750454,1075175
BC00088=318263,750454,1075175
BC00089=318263,750454,1075175
BC00090=318263,750454,1075175
BC00091=318263,750454,1075175
BC00092=318263,750454,1075175
BC00093=318263,750454,1075175
BC00094=318263,750454,1075175
BC00095=377114,750454,1075175
BC00096=397814,750454,1075175
BC00097=397814,750454,1075175
BC00098=397814,750454,1075175
BC00099=397814,750454,1075175
BC00100=397814,750454,1075175
BC00101=397814,750454,1075175
BC00102=397814,750454,1075175
BC00103=397814,750454,1075175
BC00104=397814,750454,1075175
BC00105=397814,750454,1075175
BC00106=397814,750454,1075175
BC00107=397814,750454,1075175
BC00108=397814,750454,1075175
BC00109=397814,750454,1075175
BC00110=397814,750454,1075175
BC00111=397814,750454,1075175
BC00112=397814,750454,1075175
BC00113=397814,750454,1075175
BC00114=397814,750454,1075175
BC00115=397814,750454,1075175
BC00116=383090,762961,1075175
BC00117=372387,772052,1075175
BC00118=296274,836703,1075175
BC00119=296274,836703,1075175
BC00120=296274,836703,1075175
BC00121=296274,836703,1075175
BC00122=296274,836703,1075175
BC00123=296274,836703,1075175
BC00124=296274,836703,1075175
BC00125=296274,836703,1075175
BC00126=296274,836703,1075175
BC00127=296274,836703,1075175
BC00128=296274,836703,1075175
BC00129=296274,836703,1075175
BC00130=296274,836703,1075175
BC00131=312215,899988,1075175
BC00132=312215,944285,1075175
BC00133=312215,944285,1075175
BC00134=312215,944285,1075175
BC00135=312215,944285,1075175
BC00136=312215,944285,1075175
BC00137=312215,944285,1075175
BC00138=312215,944285,1075175
BC00139=312215,944285,1075175
BC00140=312215,944285,1075175
BC00141=312215,944285,1075175
BC00142=312215,944285,1075175
BC00143=259299,938961,1075175
BC00144=259299,938961,1075175
BC00145=259299,938961,1075175
BC00146=259299,938961,1075175
BC00147=259299,938961,1075175
BC00148=259299,938961,1075175
BC00149=259299,938961,1075175
BC00150=259299,938961,1075175
BC00151=259299,938961,1075175
BC00152=259299,938961,1075175
BC00153=259299,938961,1075175
BC00154=259299,938961,1075175
BC00155=211531,951911,1075175
BC00156=211531,951911,1075175
BC00157=211531,951911,1075175
BC00158=211531,951911,1075175
BC00159=211531,951911,1075175
BC00160=211531,951911,1075175
BC00161=211531,951911,1075175
BC00162=211531,951911,1075175
BC00163=211531,951911,1075175
BC00164=211531,951911,1075175
BC00165=211531,951911,1075175
BC00166=182503,951872,1075175
BC00167=184369,953383,1075175
BC00168=184369,953399,1075175
BC00169=184333,953526,1075175
BC00170=184897,956550,1075175
BC00171=184333,953526,1075175
BC00172=184751,953664,1075175
BC00173=187887,953121,1075175
BC00174=184751,953664,1075175
BC00175=178222,948378,1075175
BC00176=185204,949959,1075175
BC00177=186100,954799,1075175
BC00178=186458,956743,1075174
BC00179=186459,956752,1075175
BC00180=186578,956775,1075175
BC00181=187141,959799,1075175
BC00182=186578,956775,1075175
BC00183=185324,949999,1075175
BC00184=153081,998123,1075175
BC00185=123088,1061215,1075175
BC00186=126332,1055781,1075175
BC00187=127630,1053613,1075175
BC00188=127630,1053623,1075175
BC00189=127630,1053607,1075175
BC00190=153753,1064749,1075175
BC00191=152152,1062093,1075175
BC00192=153753,1064749,1075175
BC00193=104366,1038154,1075175
BC00194=107120,1036610,1075175
BC00195=104366,1038154,1075175
BC00196=97490,1044180,1075175
BC00197=140343,1045718,1075175
BC00198=158643,1046375,1075175
BC00199=155464,1041036,1075175
BC00200=155106,1040455,1075175
BC00201=155106,1040463,1075175
BC00202=155288,1040367,1075175
BC00203=153687,1037711,1075175
BC00204=155288,1040367,1075175
BC00205=158891,1046297,1075175
BC00206=211337,993614,1075175
BC00207=274623,983932,1075175
BC00208=371761,1043051,1075175
BC00209=371761,1043051,1075175
BC00210=371761,1043051,1075175
BC00211=371761,1043051,1075175
BC00212=371761,1043051,1075175
BC00213=371761,1043051,1075175
BC00214=371761,1043051,1075175
BC00215=371761,1043051,1075175
BC00216=371761,1043051,1075175
BC00217=371761,1043051,1075175
BC00218=371761,1043051,1075175
BC00219=371761,1043051,1075175
BC00220=371761,1043051,1075175
BC00221=371761,1043051,1075175
BC00222=371761,1043051,1075175
BC00223=314185,938855,1075175
BC00224=247671,970611,1075175
BC00225=247671,970611,1075175
BC00226=247671,970611,1075175
BC00227=247671,970611,1075175
BC00228=247671,970611,1075175
BC00229=247671,970611,1075175
BC00230=247671,970611,1075175
BC00231=247671,970611,1075175
BC00232=247671,970611,1075175
BC00233=247671,970611,1075175
BC00234=247671,970611,1075175
BC00235=247671,970611,1075175
BC00236=303037,872055,1075175
BC00237=380992,820655,1075175
BC00238=380992,820655,1075175
BC00239=380992,820655,1075175
BC00240=380992,820655,1075175
BC00241=380992,820655,1075175
BC00242=380992,820655,1075175
BC00243=380992,820655,1075175
BC00244=380992,820655,1075175
BC00245=380992,820655,1075175
BC00246=380992,820655,1075175
BC00247=380992,820655,1075175
BC00248=380992,820655,1075175
BC00249=275256,812324,1075175
BC00250=125716,897903,1075175
BC00251=125716,897903,1075175
BC00252=125716,897903,1075175
BC00253=125716,897903,1075175
BC00254=125716,897903,1075175
BC00255=125716,897903,1075174
BC00256=125716,897903,1075171
BC00257=125716,897903,1075175
BC00258=125716,897903,1075175
BC00259=125716,897903,1075175
BC00260=125716,897903,1075175
BC00261=125716,897903,1075175
BC00262=125716,897903,1075175
BC00263=325019,822543,1075229
BC00264=325019,822543,1075229
BC00265=325019,822543,1075229
BC00266=325019,822543,1075229
BC00267=325019,822543,1075229
BC00268=325019,822543,1075229
BC00269=325019,822543,1075229
BC00270=325019,822543,1075229
BC00271=325019,822543,1075229
BC00272=325019,822543,1075229
BC00273=325019,822543,1075229
BC00274=325019,822543,1075229
BC00275=240667,871930,1075210
BC00276=81335,965219,1075175
BC00277=81335,965219,1075175
BC00278=81335,965219,1075175
BC00279=81335,965219,1075175
BC00280=81335,965219,1075175
BC00281=81335,965219,1075175
BC00282=81335,965219,1075175
BC00283=81335,965219,1075175
BC00284=39891,972466,1075175
BC00285=39891,972466,1075175
BC00286=39891,972466,1075175
BC00287=39891,972466,1075175
BC00288=39891,972466,1075175
BC00289=39891,972466,1075175
BC00290=39891,972466,1075175
BC00291=39891,972466,1075175
BC00292=126064,942124,1075175
BC00293=145718,951183,1075175
BC00294=145718,951183,1075175
BC00295=145718,951183,1075175
BC00296=145718,951183,1075175
BC00297=145718,951183,1075175
BC00298=145718,951183,1075175
BC00299=145718,951183,1075175
BC00300=145718,951183,1075175
BC00301=145718,951183,1075175
BC00302=145718,951183,1075175
BC00303=145718,951183,1075175
BC00304=145718,951183,1075175
BC00305=127193,914007,1075175
BC00306=75497,867475,1075175
BC00307=75497,867475,1075175
BC00308=75497,867475,1075175
BC00309=75497,867475,1075175
BC00310=75497,867475,1075175
BC00311=75497,867475,1075175
BC00312=75497,867475,1075175
BC00313=75497,867475,1075175
BC00314=75497,867475,1075175
BC00315=75497,867475,1075175
BC00316=75497,867475,1075175
BC00317=75497,867475,1075175
BC00318=75497,867475,1075175
BC00319=75497,867475,1075175
BC00320=75497,867475,1075175
BC00321=75497,867475,1075175
BC00322=75497,867475,1075175
BC00323=58830,852413,1075175
BC00324=43274,838354,1075175
BC00325=43274,838354,1075175
BC00326=43274,838354,1075175
BC00327=43274,838354,1075175
BC00328=43274,838354,1075175
BC00329=43274,838354,1075175
BC00330=43274,838354,1075175
BC00331=43274,838354,1075175
BC00332=43274,838354,1075175
BC00333=191439,896290,1075175
BC00334=209593,874493,1075175
BC00335=209593,874493,1075175
BC00336=209593,874493,1075175
BC00337=209593,874493,1075171
BC00338=209593,874493,1075175
BC00339=209593,874493,1075175
BC00340=209216,850926,1075175
BC00341=226866,854473,1075175
BC00342=228835,855864,1075175
BC00343=228835,855864,1075175
BC00344=228834,855864,1075173
BC00345=228834,855864,1075173
BC00346=228835,855864,1075175
BC00347=228835,855864,1075175
BC00348=228835,855864,1075175
BC00349=228835,855864,1075175
BC00350=228835,855864,1075175
BC00351=212683,986357,1075175
BC00352=212683,1004517,1075175
BC00353=212247,999872,1075175
BC00354=212146,998778,1075171
BC00355=214955,996593,1075174
BC00356=222186,994128,1075175
BC00357=222622,998773,1075175
BC00358=293477,973063,1075175
BC00359=293477,973063,1075175
BC00360=293477,973063,1075175
BC00361=293477,973063,1075175
BC00362=293477,973063,1075175
BC00363=293477,973063,1075175
BC00364=293477,973063,1075175
BC00365=293477,973063,1075175
BC00366=248777,974412,1075175
BC00367=147624,1017934,1075175
BC00368=124950,1033375,1075175
BC00369=124950,1033375,1075175
BC00370=124950,1033375,1075175
BC00371=124950,1033375,1075175
BC00372=124950,1033375,1075175
BC00373=124950,1033375,1075175
BC00374=106678,1046165,1075175
BC00375=106678,1046165,1075175
BC00376=106678,1046165,1075175
BC00377=106678,1046165,1075175
BC00378=106678,1046165,1075175
BC00379=106678,1046165,1075175
BC00380=106678,1034404,1075175
BC00381=288363,951317,1075175
BC00382=319880,932288,1075175
BC00383=316203,930177,1075175
BC00384=314732,929332,1075175
BC00385=314732,929332,1075175
BC00386=294141,940882,1075175
BC00387=285351,949486,1075175
BC00388=280844,953897,1075175
BC00389=254356,968931,1075172
BC00390=253996,970793,1075175
BC00391=256777,973747,1075175
BC00392=224914,994659,1075175
BC00393=193407,1014756,1075175
BC00394=196552,1009267,1075175
BC00395=197065,1008372,1075175
BC00396=197397,1007797,1075175
BC00397=196552,1009278,1075175
BC00398=193407,1014766,1075175
BC00399=170876,1031134,1075175
BC00400=153007,1044116,1075175
BC00401=153007,1044116,1075175
BC00402=155599,1038213,1075175
BC00403=156636,1035851,1075175
BC00404=230598,1025728,1075175
BC00405=176896,1055708,1075175
BC00406=225377,1010635,1075175
BC00407=228184,1010601,1075175
BC00408=235201,1010515,1075175
BC00409=242597,980334,1075175
BC00410=282680,816770,1075175
BC00411=287393,774165,1075175
BC00412=293866,776192,1075175
BC00413=296455,777002,1075175
BC00414=296337,777088,1075175
BC00415=296308,777110,1075175
BC00416=296189,777197,1075175
BC00417=293600,776386,1075175
BC00418=287127,774359,1075175
BC00419=265173,805126,1075175
BC00420=271841,806848,1075175
BC00421=274508,807537,1075175
BC00422=274508,807537,1075175
BC00423=271842,806893,1075175
BC00424=265174,805171,1075175
BC00425=347775,809657,1075175
BC00426=348436,809459,1075175
BC00427=348700,809380,1075175
BC00428=352833,807067,1075175
BC00429=364813,800347,1075175
BC00430=368942,798027,1075175
BC00431=368677,798106,1075175
BC00432=368016,798304,1075175
BC00433=368016,798304,1075175
BC00434=391344,687000,1075175
BC00435=391344,687000,1075175
BC00436=391344,687000,1075175
BC00437=391344,687000,1075175
BC00438=391344,687000,1075175
BC00439=391344,687000,1075175
BC00440=391344,687000,1075175
BC00441=391344,687000,1075175
BC00442=391344,687000,1075175
BC00443=391344,687000,1075175
BC00444=391344,687000,1075175
BC00445=391344,687000,1075175
BC00446=358873,687000,1075175
BC00447=250171,896024,1075175
BC00448=255370,893912,1075175
BC00449=257449,893067,1075175
BC00450=259851,897051,1075175
BC00451=270502,914711,1075175
BC00452=268422,915555,1075175
BC00453=263223,917668,1075175
BC00454=251695,824506,1075175
BC00455=253916,829548,1075175
BC00456=254804,831565,1075175
BC00457=231448,844598,1075175
BC00458=231448,844598,1075175
BC00459=189878,862044,1075175
BC00460=188570,860127,1075175
BC00461=185301,855336,1075175
BC00462=261332,833542,1075175
BC00463=297112,823286,1075175
BC00464=293523,829343,1075175
BC00465=292087,831765,1075175
BC00466=292088,831788,1075175
BC00467=293523,829365,1075175
BC00468=297112,823308,1075175
BC00469=297112,823286,1075175
BC00470=112345,954746,1075175
BC00471=112345,954746,1075175
BC00472=111546,959512,1075175
BC00473=111226,961418,1075175
BC00474=63698,969650,1075175
BC00475=64018,967744,1075175
BC00476=64817,962978,1075175
BC00477=55529,859309,1075175
BC00478=51595,858048,1075175
BC00479=50021,857544,1075175
BC00480=45895,833192,1075175
BC00481=46071,849801,1075175
BC00482=43912,844296,1075175
BC00483=45475,843733,1075175
BC00484=45475,843733,1075175
BC00485=45475,843733,1075175
BC00486=45475,843733,1075175
BC00487=45475,843733,1075175
BC00488=49382,842326,1075175
BC00489=32191,855540,1075175
BC00490=35199,856902,1075175
BC00491=36402,857447,1075175
BC00492=24170,872455,1075175
BC00493=24116,855865,1075175
BC00494=17601,856883,1075175
BC00495=10106,858388,1075175
BC00496=7107,859694,1075175
BC00497=124165,958731,1075175
BC00498=124477,964204,1075175
BC00499=124602,966393,1075175
BC00500=119899,967208,1075175
BC00501=114659,968116,1075175
BC00502=114534,965927,1075175
BC00503=114222,960453,1075175
BC00504=169497,963360,1075175
BC00505=218455,965934,1075175
BC00506=214431,967961,1075175
BC00507=212822,968772,1075175
BC00508=212822,968772,1075175
BC00509=212822,968772,1075175
BC00510=212822,968772,1075175
BC00511=218344,963319,1075175
BC00512=222368,961291,1075175
BC00513=147324,958268,1075175
BC00514=86350,984014,1075175
BC00515=90717,985390,1075175
BC00516=92241,985755,1075175
BC00517=87949,982178,1075175
BC00518=87949,982178,1075175
BC00519=87949,982178,1075175
BC00520=86202,981627,1075175
BC00521=81835,980250,1075175
BC00522=86350,984014,1075175
BC00523=118186,882849,1075175
BC00524=118313,879045,1075175
BC00525=118363,877523,1075175
BC00526=127351,877496,1075175
BC00527=127300,879018,1075175
BC00528=127173,882822,1075175
BC00529=149531,895732,1075175
BC00530=148249,891267,1075175
BC00531=148034,889482,1075175
BC00532=151775,889498,1075175
BC00533=152288,891284,1075175
BC00534=153569,895750,1075175
BC00535=119302,902119,1075175
BC00536=119440,897649,1075175
BC00537=119495,895861,1075175
BC00538=115974,895890,1075175
BC00539=115919,897678,1075175
BC00540=115781,902148,1075175
BC00541=206850,915693,1075175
BC00542=246637,921611,1075175
BC00543=251241,924622,1075175
BC00544=253082,925827,1075175
BC00545=305626,902567,1075175
BC00546=289523,905356,1075175
BC00547=289523,905356,1075175
BC00548=265997,901694,1075172
BC00549=265782,900020,1075175
BC00550=265246,895833,1075175
BC00551=152805,918674,1075175
BC00552=155644,922700,1075175
BC00553=156780,924310,1075175
BC00554=187141,913105,1075175
BC00555=135499,922155,1075175
BC00556=202417,924491,1075175
BC00557=204603,922909,1075175
BC00558=210067,918954,1075175
BC00559=285493,836258,1075175
BC00560=322674,778579,1075175
BC00561=322674,778579,1075175
BC00562=322674,778579,1075175
BC00563=322674,778579,1075175
BC00564=322674,778579,1075175
BC00565=322674,778579,1075175
BC00566=322674,778579,1075175
BC00567=322674,778579,1075175
BC00568=272555,769164,1075175
BC00569=266479,768023,1075175
BC00570=266479,768023,1075175
BC00571=267479,770239,1071365
BC00572=266799,769335,1075175
BC00573=266479,768023,1075175
BC00574=266479,768023,1075175
BC00575=266479,768023,1075175
BC00576=266479,768023,1075175
BC00577=235984,786404,1075175
BC00578=235984,786404,1075175
BC00579=235984,786404,1075175
BC00580=235984,786404,1075175
BC00581=235984,786404,1075175
BC00582=235984,786404,1075175
BC00583=235984,786404,1075175
BC00584=235984,786404,1075175
BC00585=237203,787368,1075175
BC00586=295022,827394,1075175
BC00587=205701,931185,1075175
BC00588=204812,932218,1075175
BC00589=205671,937629,1075175
BC00590=206015,939793,1075175
BC00591=202546,941762,1075175
BC00592=218293,952795,1075175
BC00593=218466,950486,1075175
BC00594=218898,944716,1075175
BC00595=188226,925402,1075175
BC00596=189298,932104,1075175
BC00597=189728,934784,1075175
BC00598=185375,937227,1075175
BC00599=184946,934546,1075175
BC00600=183874,927845,1075175
BC00601=163256,940528,1075175
BC00602=166760,944877,1075175
BC00603=168161,946617,1075175
BC00604=172960,943924,1075175
BC00605=171559,942185,1075175
BC00606=168055,937836,1075175
BC00607=205604,952176,1075175
BC00608=237375,964309,1075175
BC00609=234858,970014,1075175
BC00610=233851,972296,1075175
BC00611=237408,970622,1075175
BC00612=238426,968449,1075175
BC00613=241139,962660,1075175
BC00614=186195,958850,1075175
BC00615=137530,955476,1075175
BC00616=142340,959691,1075175
BC00617=135217,966057,1075175
BC00618=135217,966057,1075175
BC00619=134381,966543,1075175
BC00620=132263,964948,1075175
BC00621=126968,960962,1075175
BC00622=137530,955476,1075175
BC00623=284870,850327,1075175
BC00624=323104,941595,1075175
BC00625=324436,944989,1075175
BC00626=324969,946346,1075175
BC00627=379859,936839,1075175
BC00628=379326,935482,1075175
BC00629=377994,932088,1075175
BC00630=387025,925803,1075175
BC00631=391871,922431,1075175
BC00632=387133,926188,1075175
BC00633=385238,927691,1075175
BC00634=381091,925537,1075175
BC00635=365308,912570,1075175
BC00636=363166,908743,1075175
BC00637=364796,906869,1075175
BC00638=368870,902183,1075175
BC00639=358157,902408,1075175
BC00640=354876,908652,1075175
BC00641=353564,911150,1075175
BC00642=349138,907302,1075175
BC00643=357572,916934,1075175
BC00644=359178,914754,1075175
BC00645=363193,909304,1075175
BC00646=322758,853588,1075175
BC00647=135439,955204,1075175
BC00648=139952,957848,1075175
BC00649=141757,958906,1075175
BC00650=133040,997822,1075175
BC00651=133065,977483,1075175
BC00652=144047,1040883,1075175
BC00653=142698,1043050,1075175
BC00654=139327,1048468,1075175
BC00655=142698,1043050,1075175
BC00656=21214,672831,1075175
BC00657=21214,672831,429902
BC00658=66815,724118,419761
BC00659=110240,772957,337669
BC00660=124996,789553,122283
BC00661=124996,789553,122283
BC00662=124996,789553,122283
BC00663=124996,789553,122283
BC00664=124996,789553,122283
BC00665=124996,789553,122283
BC00666=124996,789553,122283
BC00667=124996,789553,122283
BC00668=124996,789553,122283
BC00669=124996,789553,122283
BC00670=124996,789553,122283
BC00671=124996,789553,122283
BC00672=124996,789553,122283
BC00673=124996,789553,122283
BC00674=124996,789553,122283
BC00675=136729,789553,283981
BC00676=136729,789553,283981
BC00677=136729,789553,283981
BC00678=136729,789553,283981
BC00679=136729,789553,283981
BC00680=136729,789553,283981
BC00681=136729,789553,283981
BC00682=136729,789553,283981
BC00683=136729,789553,283981
BC00684=136729,789553,283981
BC00685=163194,789553,386705
BC00686=163194,789553,386705
BC00687=163194,789553,386705
BC00688=163194,789553,386705
BC00689=163194,789553,386705
BC00690=163194,789553,386705
BC00691=163194,789553,386705
BC00692=163194,789553,386705
BC00693=163194,789553,386705
BC00694=163194,789553,386705
BC00695=110240,772957,337669
BC00696=66815,724118,419761
BC00697=66815,670858,419761
BC00698=252765,670858,277331
BC00699=322808,760288,131711
BC00700=322808,760288,131711
BC00701=322808,760288,131711
BC00702=322808,760288,131711
BC00703=322808,760288,131711
BC00704=322808,760288,131711
BC00705=322808,760288,131711
BC00706=322808,760288,131711
BC00707=322808,760288,131711
BC00708=335534,789553,204922
BC00709=335534,789553,204922
BC00710=335534,789553,204922
BC00711=335534,789553,204922
BC00712=335534,789553,204922
BC00713=335534,789553,204922
BC00714=335534,789553,204922
BC00715=335534,789553,204922
BC00716=335534,789553,204922
BC00717=344006,752651,139062
BC00718=344006,752651,139062
BC00719=344006,752651,139062
BC00720=344006,752651,139062
BC00721=344006,752651,139062
BC00722=344006,752651,139062
BC00723=344006,752651,139062
BC00724=344006,752651,139062
BC00725=344006,752651,139062
BC00726=300933,750795,218908
BC00727=283893,750061,250495
BC00728=276320,749735,264534
BC00729=276320,749735,264534
BC00730=276320,749735,264534
BC00731=276320,749735,264534
BC00732=276320,749735,264534
BC00733=276320,749735,264534
BC00734=276320,749735,264534
BC00735=276320,749735,264534
BC00736=276320,749735,264534
BC00737=248857,763770,138691
BC00738=248857,763770,138691
BC00739=248857,763770,138691
BC00740=248857,763770,138691
BC00741=248857,763770,138691
BC00742=248857,763770,138691
BC00743=248857,763770,138691
BC00744=248857,763770,138691
BC00745=248857,763770,138691
BC00746=287864,789553,132710
BC00747=287864,789553,132710
BC00748=287864,789553,132710
BC00749=287864,789553,132710
BC00750=287864,789553,132710
BC00751=287864,789553,132710
BC00752=287864,789553,132710
BC00753=287864,789553,132710
BC00754=287864,789553,132710
BC00755=287864,789553,132710
BC00756=287864,789553,132710
BC00757=287864,789553,132710
BC00758=279829,789553,53
BC00759=279829,789553,53
BC00760=279829,789553,53
BC00761=279829,789553,53
BC00762=279829,789553,53
BC00763=279829,789553,53
BC00764=279829,789553,53
BC00765=279829,789553,53
BC00766=279829,789553,53
BC00767=279829,789553,53
BC00768=279829,789553,53
BC00769=279829,789553,53
BC00770=279829,789553,53
BC00771=312324,789553,158805
BC00772=312324,789553,158805
BC00773=312324,789553,158804
BC00774=312324,789553,158805
BC00775=312324,789553,158805
BC00776=312324,789553,158805
BC00777=303082,768394,105099
BC00778=303082,768394,105099
BC00779=303082,768394,105099
BC00780=303082,768394,105099
BC00781=303082,768394,105099
BC00782=303082,768394,105099
BC00783=287868,781442,183325
BC00784=278410,789553,231953
BC00785=278410,789553,231953
BC00786=278410,789553,231953
BC00787=278410,789553,231953
BC00788=278410,789553,231953
BC00789=278410,789553,231953
BC00790=283893,750061,250495
BC00791=300933,750795,218908
BC00792=376723,772526,120737
BC00793=376723,772526,120737
BC00794=376723,772526,120737
BC00795=376723,772526,120737
BC00796=376723,772526,120737
BC00797=376723,772526,120737
BC00798=385013,737075,95404
BC00799=385013,737075,95404
BC00800=385013,737075,95404
BC00801=385013,737075,95404
BC00802=385013,737075,95404
BC00803=385013,737075,95404
BC00804=365962,760163,122379
BC00805=365962,760163,122379
BC00806=365962,760163,122379
BC00807=365962,760163,122379
BC00808=365962,760163,122379
BC00809=365962,760163,122379
BC00810=365962,760163,122379
BC00811=252765,670858,277331
BC00812=66815,670858,419761
BC00813=66815,724118,419761
BC00814=110240,772957,337669
BC00815=118803,789553,240458
BC00816=118803,789553,240458
BC00817=118803,789553,240458
BC00818=118803,789553,240458
BC00819=118803,789553,240458
BC00820=118803,789553,240458
BC00821=130259,789553,198376
BC00822=110709,789553,198376
BC00823=113251,789553,198376
BC00824=113251,789553,198376
BC00825=113251,789553,198376
BC00826=113251,789553,198376
BC00827=113251,789553,198376
BC00828=113251,789553,198376
BC00829=113251,789553,198376
BC00830=113251,789553,198376
BC00831=113251,789553,198376
BC00832=113251,789553,198376
BC00833=113251,789553,198376
BC00834=113251,789553,198376
BC00835=113251,789553,198376
BC00836=113251,789553,228042
BC00837=113251,789553,280292
BC00838=113251,789553,280290
BC00839=113251,789553,280290
BC00840=113251,789553,280290
BC00841=113251,789553,280290
BC00842=113251,789553,280290
BC00843=113251,789553,280290
BC00844=113251,789553,280290
BC00845=110240,772957,337669
BC00846=66815,724118,419761
BC00847=66815,670858,419761
BC00848=252765,670858,277331
BC00849=298333,782774,240815
BC00850=298333,782774,240815
BC00851=298333,782774,240815
BC00852=298333,782774,240815
BC00853=298333,782774,240815
BC00854=298333,782774,240815
BC00855=277596,773081,190929
BC00856=277596,773081,190929
BC00857=277596,773081,190929
BC00858=277596,773081,190929
BC00859=277596,773081,190929
BC00860=277596,773081,190929
BC00861=252765,670858,277331
BC00862=66815,670858,419761
BC00863=66815,724118,419761
BC00864=110240,772957,337669
BC00865=116545,789553,319269
BC00866=116545,789553,319269
BC00867=116545,789553,319269
BC00868=116545,789553,319269
BC00869=116545,789553,319269
BC00870=116545,789553,319269
BC00871=104258,789553,379308
BC00872=104258,789553,379308
BC00873=104258,789553,379308
BC00874=104258,789553,379308
BC00875=104258,789553,379308
BC00876=104258,789553,379308
BC00877=110240,772957,337669
BC00878=66815,724118,419761
BC00879=66815,670858,419761
BC00880=252765,670858,277331
BC00881=286674,787255,240962
BC00882=286675,787255,240962
BC00883=286675,787255,240962
BC00884=286675,787255,240962
BC00885=286674,787255,240962
BC00886=286674,787255,240962
BC00887=267109,758037,158941
BC00888=267109,758037,158941
BC00889=267109,758037,158941
BC00890=267109,758037,158941
BC00891=267109,758037,158941
BC00892=267109,758037,158941
BC00893=283893,750061,250495
BC00894=360336,760725,110934
BC00895=360336,760725,110934
BC00896=360336,760725,110934
BC00897=360336,760725,110934
BC00898=360336,760725,110934
BC00899=360336,760725,110934
BC00900=371149,789553,191296
BC00901=371149,789553,191296
BC00902=371149,789553,191296
BC00903=371149,789553,191296
BC00904=371149,789553,191296
BC00905=371149,789553,191296
BC00906=283893,750061,250495
BC00907=292970,789553,136523
BC00908=292970,789553,136523
BC00909=292970,789553,136523
BC00910=292970,789553,136523
BC00911=292970,789553,136523
BC00912=292970,789552,136519
BC00913=292970,789553,136523
BC00914=292970,789553,136523
BC00915=256495,759418,21571
BC00916=256495,759418,21571
BC00917=256495,759418,21571
BC00918=256495,759418,21571
BC00919=256495,759418,21571
BC00920=256495,759418,21571
BC00921=256075,748610,41729
BC00922=255916,738170,60084
BC00923=255916,738170,60084
BC00924=255916,738170,60084
BC00925=255916,738170,60084
BC00926=255916,738170,60084
BC00927=255916,738170,60084
BC00928=262339,748900,193466
BC00929=165820,667836,534036
BC00930=21214,672831,1075175
EC00000=798156,1112951
EC00001=798156,1112951
EC00002=798156,1112951
EC00003=798156,1112951
EC00004=798156,1112951
EC00005=798156,1112951
EC00006=798156,1112951
EC00007=798156,1112951
EC00008=798156,1112951
EC00009=798156,1112951
EC00010=798156,1112951
EC00011=798156,1112951
EC00012=798156,1112951
EC00013=798156,1112951
EC00014=798156,1112951
EC00015=798156,1112951
EC00016=798156,1112951
EC00017=798156,1112951
EC00018=798156,1112951
EC00019=798156,1112951
EC00020=798156,1112951
EC00021=798156,1112951
EC00022=798156,1112951
EC00023=798156,1112951
EC00024=798156,1112951
EC00025=798156,1112951
EC00026=798156,1112951
EC00027=798156,1112951
EC00028=798156,1112951
EC00029=798156,1112951
EC00030=798156,1112951
EC00031=798156,1112951
EC00032=798156,1112951
EC00033=798156,1112951
EC00034=798156,1112951
EC00035=798155,1112950
EC00036=798155,1112950
EC00037=798155,1112950
EC00038=798154,1112949
EC00039=798154,1112949
EC00040=798154,1112949
EC00041=798154,1112949
EC00042=798154,1112949
EC00043=798153,1112949
EC00044=798156,1112951
EC00045=798156,1112951
EC00046=798156,1112951
EC00047=798156,1112951
EC00048=798156,1112951
EC00049=798156,1112951
EC00050=798156,1112951
EC00051=798156,1112951
EC00052=798156,1112951
EC00053=798156,1112951
EC00054=798156,1112951
EC00055=798156,1112951
EC00056=798156,1112951
EC00057=798156,1112951
EC00058=798156,1112951
EC00059=798156,1112951
EC00060=798156,1112951
EC00061=798156,1112951
EC00062=798156,1112951
EC00063=798156,1112951
EC00064=798155,1112950
EC00065=798155,1112950
EC00066=798156,1112951
EC00067=798156,1112951
EC00068=798156,1112951
EC00069=798156,1112951
EC00070=798156,1112951
EC00071=798156,1112951
EC00072=798156,1112951
EC00073=798156,1112951
EC00074=798156,1112951
EC00075=798156,1112951
EC00076=798156,1112951
EC00077=798156,1112951
EC00078=798156,1112951
EC00079=798156,1112951
EC00080=798156,1112951
EC00081=798156,1112951
EC00082=798156,1112951
EC00083=798156,1112951
EC00084=798156,1112951
EC00085=798156,1112951
EC00086=798156,1112951
EC00087=798156,1112951
EC00088=798156,1112951
EC00089=798156,1112951
EC00090=798156,1112951
EC00091=798156,1112951
EC00092=798156,1112951
EC00093=798156,1112951
EC00094=798156,1112951
EC00095=798156,1112951
EC00096=798156,1112951
EC00097=798156,1112951
EC00098=798156,1112951
EC00099=798156,1112951
EC00100=798156,1112951
EC00101=798156,1112951
EC00102=798156,1112951
EC00103=798156,1112951
EC00104=798156,1112951
EC00105=798156,1112951
EC00106=798156,1112951
EC00107=798156,1112951
EC00108=798156,1112951
EC00109=798156,1112951
EC00110=798156,1112951
EC00111=798156,1112951
EC00112=798156,1112951
EC00113=798156,1112951
EC00114=798156,1112951
EC00115=798156,1112951
EC00116=798156,1112951
EC00117=798156,1112951
EC00118=798156,1112951
EC00119=798156,1112951
EC00120=798156,1112951
EC00121=798156,1112951
EC00122=798156,1112951
EC00123=798156,1112951
EC00124=798156,1112951
EC00125=798156,1112951
EC00126=798156,1112951
EC00127=798156,1112951
EC00128=798156,1112951
EC00129=798156,1112951
EC00130=798156,1112951
EC00131=798156,1112951
EC00132=798156,1112951
EC00133=798156,1112951
EC00134=798156,1112951
EC00135=798156,1112951
EC00136=798156,1112951
EC00137=798156,1112951
EC00138=798156,1112951
EC00139=798156,1112951
EC00140=798156,1112951
EC00141=798156,1112951
EC00142=798156,1112951
EC00143=798156,1112951
EC00144=798156,1112951
EC00145=798156,1112951
EC00146=798156,1112951
EC00147=798156,1112951
EC00148=798156,1112951
EC00149=798156,1112951
EC00150=798156,1112951
EC00151=798156,1112951
EC00152=798156,1112951
EC00153=798156,1112951
EC00154=798156,1112951
EC00155=798156,1112951
EC00156=798156,1112951
EC00157=798156,1112951
EC00158=798156,1112951
EC00159=798156,1112951
EC00160=798156,1112951
EC00161=798156,1112951
EC00162=798156,1112951
EC00163=798156,1112951
EC00164=798156,1112951
EC00165=798156,1112951
EC00166=798156,1112951
EC00167=798156,1112951
EC00168=798156,1112951
EC00169=798156,1112951
EC00170=798156,1112951
EC00171=798156,1112951
EC00172=798156,1112951
EC00173=798156,1112951
EC00174=798156,1112951
EC00175=798156,1112951
EC00176=798156,1112951
EC00177=798156,1112951
EC00178=798155,1112950
EC00179=798156,1112951
EC00180=798156,1112951
EC00181=798156,1112951
EC00182=798156,1112951
EC00183=798156,1112951
EC00184=798156,1112951
EC00185=798156,1112951
EC00186=798156,1112951
EC00187=798156,1112951
EC00188=798156,1112951
EC00189=798156,1112951
EC00190=798156,1112951
EC00191=798156,1112951
EC00192=798156,1112951
EC00193=798156,1112951
EC00194=798156,1112951
EC00195=798156,1112951
EC00196=798156,1112951
EC00197=798156,1112951
EC00198=798156,1112951
EC00199=798156,1112951
EC00200=798156,1112951
EC00201=798156,1112951
EC00202=798156,1112951
EC00203=798156,1112951
EC00204=798156,1112951
EC00205=798156,1112951
EC00206=798156,1112951
EC00207=798156,1112951
EC00208=798156,1112951
EC00209=798156,1112951
EC00210=798156,1112951
EC00211=798156,1112951
EC00212=798156,1112951
EC00213=798156,1112951
EC00214=798156,1112951
EC00215=798156,1112951
EC00216=798156,1112951
EC00217=798156,1112951
EC00218=798156,1112951
EC00219=798156,1112951
EC00220=798156,1112951
EC00221=798156,1112951
EC00222=798156,1112951
EC00223=798156,1112951
EC00224=798156,1112951
EC00225=798156,1112951
EC00226=798156,1112951
EC00227=798156,1112951
EC00228=798156,1112951
EC00229=798156,1112951
EC00230=798156,1112951
EC00231=798156,1112951
EC00232=798156,1112951
EC00233=798156,1112951
EC00234=798156,1112951
EC00235=798156,1112951
EC00236=798156,1112951
EC00237=798156,1112951
EC00238=798156,1112951
EC00239=798156,1112951
EC00240=798156,1112951
EC00241=798156,1112951
EC00242=798156,1112951
EC00243=798156,1112951
EC00244=798156,1112951
EC00245=798156,1112951
EC00246=798156,1112951
EC00247=798156,1112951
EC00248=798156,1112951
EC00249=798156,1112951
EC00250=798156,1112951
EC00251=798156,1112951
EC00252=798156,1112951
EC00253=798156,1112951
EC00254=798156,1112951
EC00255=798156,1112951
EC00256=798155,1112951
EC00257=798156,1112951
EC00258=798156,1112951
EC00259=798156,1112951
EC00260=798156,1112951
EC00261=798156,1112951
EC00262=798156,1112951
EC00263=798156,1112951
EC00264=798156,1112951
EC00265=798156,1112951
EC00266=798156,1112951
EC00267=798156,1112951
EC00268=798156,1112951
EC00269=798156,1112951
EC00270=798156,1112951
EC00271=798156,1112951
EC00272=798156,1112951
EC00273=798156,1112951
EC00274=798156,1112951
EC00275=798156,1112951
EC00276=798156,1112951
EC00277=798156,1112951
EC00278=798156,1112951
EC00279=798156,1112951
EC00280=798156,1112951
EC00281=798156,1112951
EC00282=798156,1112951
EC00283=798156,1112951
EC00284=798156,1112951
EC00285=798156,1112951
EC00286=798156,1112951
EC00287=798156,1112951
EC00288=798156,1112951
EC00289=798156,1112951
EC00290=798156,1112951
EC00291=798156,1112951
EC00292=798156,1112951
EC00293=798156,1112951
EC00294=798156,1112951
EC00295=798156,1112951
EC00296=798156,1112951
EC00297=798156,1112951
EC00298=798156,1112951
EC00299=798156,1112951
EC00300=798156,1112951
EC00301=798156,1112951
EC00302=798156,1112951
EC00303=798156,1112951
EC00304=798156,1112951
EC00305=798156,1112951
EC00306=798156,1112951
EC00307=798156,1112951
EC00308=798156,1112951
EC00309=798156,1112951
EC00310=798156,1112951
EC00311=798156,1112951
EC00312=798156,1112951
EC00313=798156,1112951
EC00314=798156,1112951
EC00315=798156,1112951
EC00316=798156,1112951
EC00317=798156,1112951
EC00318=798156,1112951
EC00319=798156,1112951
EC00320=798156,1112951
EC00321=798156,1112951
EC00322=798156,1112951
EC00323=798156,1112951
EC00324=798156,1112951
EC00325=798156,1112951
EC00326=798156,1112951
EC00327=798156,1112951
EC00328=798156,1112951
EC00329=798156,1112951
EC00330=798156,1112951
EC00331=798156,1112951
EC00332=798156,1112951
EC00333=798156,1112951
EC00334=798156,1112951
EC00335=798156,1112951
EC00336=798156,1112951
EC00337=798155,1112950
EC00338=798156,1112951
EC00339=798156,1112951
EC00340=798156,1112951
EC00341=798156,1112951
EC00342=798156,1112951
EC00343=798156,1112951
EC00344=798155,1112951
EC00345=798155,1112951
EC00346=798156,1112951
EC00347=798156,1112951
EC00348=798156,1112951
EC00349=798156,1112951
EC00350=798156,1112951
EC00351=798156,1112951
EC00352=798156,1112951
EC00353=798156,1112951
EC00354=798155,1112950
EC00355=798156,1112951
EC00356=798156,1112951
EC00357=798156,1112951
EC00358=798156,1112951
EC00359=798156,1112951
EC00360=798156,1112951
EC00361=798156,1112951
EC00362=798156,1112951
EC00363=798156,1112951
EC00364=798156,1112951
EC00365=798156,1112951
EC00366=798156,1112951
EC00367=798156,1112951
EC00368=798156,1112951
EC00369=798156,1112951
EC00370=798156,1112951
EC00371=798156,1112951
EC00372=798156,1112951
EC00373=798156,1112951
EC00374=798156,1112951
EC00375=798156,1112951
EC00376=798156,1112951
EC00377=798156,1112951
EC00378=798156,1112951
EC00379=798156,1112951
EC00380=798156,1112951
EC00381=798156,1112951
EC00382=798156,1112951
EC00383=798156,1112951
EC00384=798156,1112951
EC00385=798156,1112951
EC00386=798156,1112951
EC00387=798156,1112951
EC00388=798156,1112951
EC00389=798155,1112950
EC00390=798156,1112951
EC00391=798156,1112951
EC00392=798156,1112951
EC00393=798156,1112951
EC00394=798156,1112951
EC00395=798156,1112951
EC00396=798156,1112951
EC00397=798156,1112951
EC00398=798156,1112951
EC00399=798156,1112951
EC00400=798156,1112951
EC00401=798156,1112951
EC00402=798156,1112951
EC00403=798156,1112951
EC00404=798156,1112951
EC00405=798156,1112951
EC00406=798156,1112951
EC00407=798156,1112951
EC00408=798156,1112951
EC00409=798156,1112951
EC00410=798156,1112951
EC00411=798156,1112951
EC00412=798156,1112951
EC00413=798156,1112951
EC00414=798156,1112951
EC00415=798156,1112951
EC00416=798156,1112951
EC00417=798156,1112951
EC00418=798156,1112951
EC00419=798156,1112951
EC00420=798156,1112951
EC00421=798156,1112951
EC00422=798156,1112951
EC00423=798156,1112951
EC00424=798156,1112951
EC00425=798156,1112951
EC00426=798156,1112951
EC00427=798156,1112951
EC00428=798156,1112951
EC00429=798156,1112951
EC00430=798156,1112951
EC00431=798156,1112951
EC00432=798156,1112951
EC00433=798156,1112951
EC00434=798156,1112951
EC00435=798156,1112951
EC00436=798156,1112951
EC00437=798156,1112951
EC00438=798156,1112951
EC00439=798156,1112951
EC00440=798156,1112951
EC00441=798156,1112951
EC00442=798156,1112951
EC00443=798156,1112951
EC00444=798156,1112951
EC00445=798156,1112951
EC00446=798156,1112951
EC00447=798156,1112951
EC00448=798156,1112951
EC00449=798156,1112951
EC00450=798156,1112951
EC00451=798156,1112951
EC00452=798156,1112951
EC00453=798156,1112951
EC00454=798156,1112951
EC00455=798156,1112951
EC00456=798156,1112951
EC00457=798156,1112951
EC00458=798156,1112951
EC00459=798156,1112951
EC00460=798156,1112951
EC00461=798156,1112951
EC00462=798156,1112951
EC00463=798156,1112951
EC00464=798156,1112951
EC00465=798156,1112951
EC00466=798156,1112951
EC00467=798156,1112951
EC00468=798156,1112951
EC00469=798156,1112951
EC00470=798156,1112951
EC00471=798156,1112951
EC00472=798156,1112951
EC00473=798156,1112951
EC00474=798156,1112951
EC00475=798156,1112951
EC00476=798156,1112951
EC00477=798156,1112951
EC00478=798156,1112951
EC00479=798156,1112951
EC00480=798156,1112951
EC00481=798156,1112951
EC00482=798156,1112951
EC00483=798156,1112951
EC00484=798156,1112951
EC00485=798156,1112951
EC00486=798156,1112951
EC00487=798156,1112951
EC00488=798156,1112951
EC00489=798156,1112951
EC00490=798156,1112951
EC00491=798156,1112951
EC00492=798156,1112951
EC00493=798156,1112951
EC00494=798156,1112951
EC00495=798156,1112951
EC00496=798156,1112951
EC00497=798156,1112951
EC00498=798156,1112951
EC00499=798156,1112951
EC00500=798156,1112951
EC00501=798156,1112951
EC00502=798156,1112951
EC00503=798156,1112951
EC00504=798156,1112951
EC00505=798156,1112951
EC00506=798156,1112951
EC00507=798156,1112951
EC00508=798156,1112951
EC00509=798156,1112951
EC00510=798156,1112951
EC00511=798156,1112951
EC00512=798156,1112951
EC00513=798156,1112951
EC00514=798156,1112951
EC00515=798156,1112951
EC00516=798156,1112951
EC00517=798156,1112951
EC00518=798156,1112951
EC00519=798156,1112951
EC00520=798156,1112951
EC00521=798156,1112951
EC00522=798156,1112951
EC00523=798156,1112951
EC00524=798156,1112951
EC00525=798156,1112951
EC00526=798156,1112951
EC00527=798156,1112951
EC00528=798156,1112951
EC00529=798156,1112951
EC00530=798156,1112951
EC00531=798156,1112951
EC00532=798156,1112951
EC00533=798156,1112951
EC00534=798156,1112951
EC00535=798156,1112951
EC00536=798156,1112951
EC00537=798156,1112951
EC00538=798156,1112951
EC00539=798156,1112951
EC00540=798156,1112951
EC00541=798156,1112951
EC00542=798156,1112951
EC00543=798156,1112951
EC00544=798156,1112951
EC00545=798156,1112951
EC00546=798156,1112951
EC00547=798156,1112951
EC00548=798155,1112950
EC00549=798156,1112951
EC00550=798156,1112951
EC00551=798156,1112951
EC00552=798156,1112951
EC00553=798156,1112951
EC00554=798156,1112951
EC00555=798156,1112951
EC00556=798156,1112951
EC00557=798156,1112951
EC00558=798156,1112951
EC00559=798156,1112951
EC00560=798156,1112951
EC00561=798156,1112951
EC00562=798156,1112951
EC00563=798156,1112951
EC00564=798156,1112951
EC00565=798156,1112951
EC00566=798156,1112951
EC00567=798156,1112951
EC00568=798156,1112951
EC00569=798156,1112951
EC00570=798156,1112951
EC00571=798156,1112951
EC00572=798156,1112951
EC00573=798156,1112951
EC00574=798156,1112951
EC00575=798156,1112951
EC00576=798156,1112951
EC00577=798156,1112951
EC00578=798156,1112951
EC00579=798156,1112951
EC00580=798156,1112951
EC00581=798156,1112951
EC00582=798156,1112951
EC00583=798156,1112951
EC00584=798156,1112951
EC00585=798156,1112951
EC00586=798156,1112951
EC00587=798156,1112951
EC00588=798156,1112951
EC00589=798156,1112951
EC00590=798156,1112951
EC00591=798156,1112951
EC00592=798156,1112951
EC00593=798156,1112951
EC00594=798156,1112951
EC00595=798156,1112951
EC00596=798156,1112951
EC00597=798156,1112951
EC00598=798156,1112951
EC00599=798156,1112951
EC00600=798156,1112951
EC00601=798156,1112951
EC00602=798156,1112951
EC00603=798156,1112951
EC00604=798156,1112951
EC00605=798156,1112951
EC00606=798156,1112951
EC00607=798156,1112951
EC00608=798156,1112951
EC00609=798156,1112951
EC00610=798156,1112951
EC00611=798156,1112951
EC00612=798156,1112951
EC00613=798156,1112951
EC00614=798156,1112951
EC00615=798156,1112951
EC00616=798156,1112951
EC00617=798156,1112951
EC00618=798156,1112951
EC00619=798156,1112951
EC00620=798156,1112951
EC00621=798156,1112951
EC00622=798156,1112951
EC00623=798156,1112951
EC00624=798156,1112951
EC00625=798156,1112951
EC00626=798156,1112951
EC00627=798156,1112951
EC00628=798156,1112951
EC00629=798156,1112951
EC00630=798156,1112951
EC00631=798156,1112951
EC00632=798156,1112951
EC00633=798156,1112951
EC00634=798156,1112951
EC00635=798156,1112951
EC00636=798156,1112951
EC00637=798156,1112951
EC00638=798156,1112951
EC00639=798156,1112951
EC00640=798156,1112951
EC00641=798156,1112951
EC00642=798156,1112951
EC00643=798156,1112951
EC00644=798156,1112951
EC00645=798156,1112951
EC00646=798156,1112951
EC00647=798156,1112951
EC00648=798156,1112951
EC00649=798156,1112951
EC00650=798156,1112951
EC00651=798156,1112951
EC00652=798156,1112951
EC00653=798156,1112951
EC00654=798156,1112951
EC00655=798156,1112951
EC00656=798156,1112951
EC00657=798156,1112951
EC00658=798156,1112951
EC00659=798156,1112951
EC00660=798156,1112951
EC00661=798156,1112951
EC00662=798156,1112951
EC00663=798156,1112951
EC00664=798156,1112951
EC00665=798156,1112951
EC00666=798156,1112951
EC00667=798156,1112951
EC00668=798156,1112951
EC00669=798156,1112951
EC00670=798156,1112951
EC00671=798156,1112951
EC00672=798156,1112951
EC00673=798156,1112951
EC00674=798156,1112951
EC00675=798156,1112951
EC00676=798156,1112951
EC00677=798156,1112951
EC00678=798156,1112951
EC00679=798156,1112951
EC00680=798156,1112951
EC00681=798156,1112951
EC00682=798156,1112951
EC00683=798156,1112951
EC00684=798156,1112951
EC00685=798156,1112951
EC00686=798156,1112951
EC00687=798156,1112951
EC00688=798156,1112951
EC00689=798156,1112951
EC00690=798156,1112951
EC00691=798156,1112951
EC00692=798156,1112951
EC00693=798156,1112951
EC00694=798156,1112951
EC00695=798156,1112951
EC00696=798156,1112951
EC00697=798156,1112951
EC00698=798156,1112951
EC00699=798156,1112951
EC00700=798156,1112951
EC00701=798156,1112951
EC00702=798156,1112951
EC00703=798156,1112951
EC00704=798156,1112951
EC00705=798156,1112951
EC00706=798156,1112951
EC00707=798156,1112951
EC00708=798156,1112951
EC00709=798156,1112951
EC00710=798156,1112951
EC00711=798156,1112951
EC00712=798156,1112951
EC00713=798156,1112951
EC00714=798156,1112951
EC00715=798156,1112951
EC00716=798156,1112951
EC00717=798156,1112951
EC00718=798156,1112951
EC00719=798156,1112951
EC00720=798156,1112951
EC00721=798156,1112951
EC00722=798156,1112951
EC00723=798156,1112951
EC00724=798156,1112951
EC00725=798156,1112951
EC00726=798156,1112951
EC00727=798156,1112951
EC00728=798156,1112951
EC00729=798156,1112951
EC00730=798156,1112951
EC00731=798156,1112951
EC00732=798156,1112951
EC00733=798156,1112951
EC00734=798156,1112951
EC00735=798156,1112951
EC00736=798156,1112951
EC00737=798156,1112951
EC00738=798156,1112951
EC00739=798156,1112951
EC00740=798156,1112951
EC00741=798156,1112951
EC00742=798156,1112951
EC00743=798156,1112951
EC00744=798156,1112951
EC00745=798156,1112951
EC00746=798156,1112951
EC00747=798156,1112951
EC00748=798156,1112951
EC00749=798156,1112951
EC00750=798156,1112951
EC00751=798156,1112951
EC00752=798156,1112951
EC00753=798156,1112951
EC00754=798156,1112951
EC00755=798156,1112951
EC00756=798156,1112951
EC00757=798156,1112951
EC00758=798156,1112951
EC00759=798156,1112951
EC00760=798156,1112951
EC00761=798156,1112951
EC00762=798156,1112951
EC00763=798156,1112951
EC00764=798156,1112951
EC00765=798156,1112951
EC00766=798156,1112951
EC00767=798156,1112951
EC00768=798156,1112951
EC00769=798156,1112951
EC00770=798156,1112951
EC00771=798156,1112951
EC00772=798156,1112951
EC00773=798156,1112949
EC00774=798156,1112951
EC00775=798156,1112951
EC00776=798156,1112951
EC00777=798156,1112951
EC00778=798156,1112951
EC00779=798156,1112951
EC00780=798156,1112951
EC00781=798156,1112951
EC00782=798156,1112951
EC00783=798156,1112951
EC00784=798156,1112951
EC00785=798156,1112951
EC00786=798156,1112951
EC00787=798156,1112951
EC00788=798156,1112951
EC00789=798156,1112951
EC00790=798156,1112951
EC00791=798156,1112951
EC00792=798156,1112951
EC00793=798156,1112951
EC00794=798156,1112951
EC00795=798156,1112951
EC00796=798156,1112951
EC00797=798156,1112951
EC00798=798156,1112951
EC00799=798156,1112951
EC00800=798156,1112951
EC00801=798156,1112951
EC00802=798156,1112951
EC00803=798156,1112951
EC00804=798156,1112951
EC00805=798156,1112951
EC00806=798156,1112951
EC00807=798156,1112951
EC00808=798156,1112951
EC00809=798156,1112951
EC00810=798156,1112951
EC00811=798156,1112951
EC00812=798156,1112951
EC00813=798156,1112951
EC00814=798156,1112951
EC00815=798156,1112951
EC00816=798156,1112951
EC00817=798156,1112951
EC00818=798156,1112951
EC00819=798156,1112951
EC00820=798156,1112951
EC00821=798156,1112951
EC00822=798156,1112951
EC00823=798156,1112951
EC00824=798156,1112951
EC00825=798156,1112951
EC00826=798156,1112951
EC00827=798156,1112951
EC00828=798156,1112951
EC00829=798156,1112951
EC00830=798156,1112951
EC00831=798156,1112951
EC00832=798156,1112951
EC00833=798156,1112951
EC00834=798156,1112951
EC00835=798156,1112951
EC00836=798156,1112951
EC00837=798156,1112951
EC00838=798155,1112950
EC00839=798155,1112950
EC00840=798155,1112950
EC00841=798155,1112950
EC00842=798155,1112950
EC00843=798155,1112950
EC00844=798155,1112950
EC00845=798156,1112951
EC00846=798156,1112951
EC00847=798156,1112951
EC00848=798156,1112951
EC00849=798156,1112951
EC00850=798156,1112951
EC00851=798156,1112951
EC00852=798156,1112951
EC00853=798156,1112951
EC00854=798156,1112951
EC00855=798156,1112951
EC00856=798156,1112951
EC00857=798156,1112951
EC00858=798156,1112951
EC00859=798156,1112951
EC00860=798156,1112951
EC00861=798156,1112951
EC00862=798156,1112951
EC00863=798156,1112951
EC00864=798156,1112951
EC00865=798156,1112951
EC00866=798156,1112951
EC00867=798156,1112951
EC00868=798156,1112951
EC00869=798156,1112951
EC00870=798156,1112951
EC00871=798156,1112951
EC00872=798156,1112951
EC00873=798156,1112951
EC00874=798156,1112951
EC00875=798156,1112951
EC00876=798156,1112951
EC00877=798156,1112951
EC00878=798156,1112951
EC00879=798156,1112951
EC00880=798156,1112951
EC00881=798156,1112951
EC00882=798156,1112951
EC00883=798156,1112951
EC00884=798156,1112951
EC00885=798156,1112951
EC00886=798156,1112951
EC00887=798156,1112951
EC00888=798156,1112951
EC00889=798156,1112951
EC00890=798156,1112951
EC00891=798156,1112951
EC00892=798156,1112951
EC00893=798156,1112951
EC00894=798156,1112951
EC00895=798156,1112951
EC00896=798156,1112951
EC00897=798156,1112951
EC00898=798156,1112951
EC00899=798156,1112951
EC00900=798156,1112951
EC00901=798156,1112951
EC00902=798156,1112951
EC00903=798156,1112951
EC00904=798156,1112951
EC00905=798156,1112951
EC00906=798156,1112951
EC00907=798156,1112951
EC00908=798156,1112951
EC00909=798156,1112951
EC00910=798156,1112951
EC00911=798156,1112951
EC00912=798155,1112949
EC00913=798156,1112951
EC00914=798156,1112951
EC00915=798156,1112951
EC00916=798156,1112951
EC00917=798156,1112951
EC00918=798156,1112951
EC00919=798156,1112951
EC00920=798156,1112951
EC00921=798156,1112951
EC00922=798156,1112951
EC00923=798156,1112951
EC00924=798156,1112951
EC00925=798156,1112951
EC00926=798156,1112951
EC00927=798156,1112951
EC00928=798156,1112951
EC00929=798156,1112951
EC00930=798156,1112951
///POSTYPE BASE
///RECTAN
///RCONF 0,0,0,0,0,0,0,0,0,0,0,0,0,0,0,0,0,0,0,0,0,0,0,0
P00006=0.222,-3.123,-1.508,0.0000,0.0000,0.0000
P00021=-0.225,-6.128,-0.405,0.0000,0.0000,0.0000
P00022=0.222,-3.123,-1.508,0.0000,0.0000,0.0000
P00023=0.143,-0.036,0.682,0.0000,0.0000,0.0000
P00024=0.145,-0.552,1.326,0.0000,0.0000,0.0000
P00025=-2.003,0.006,0.728,0.0000,0.0000,0.0000
P00026=0.562,-0.002,-0.337,0.0000,0.0000,0.0000
P00027=-0.746,0.015,-9.096,0.0000,0.0000,0.0000
P00028=-2.237,-0.018,-7.702,0.0000,0.0000,0.0000
P00029=-2.156,-0.086,-4.681,0.0000,0.0000,0.0000
P00030=5.926,-4.294,-1.390,0.0000,0.0000,0.0000
P00031=1.853,-0.001,-1.549,0.0000,0.0000,0.0000
P00032=1.957,0.503,-7.217,0.0000,0.0000,0.0000
///RCONF 0,0,0,0,1,0,0,0,0,0,0,0,0,0,0,0,0,0,0,0,0,0,0,0
P00033=-0.123,0.612,-5.012,0.0000,0.0000,0.0000
///RCONF 0,0,0,0,0,0,0,0,0,0,0,0,0,0,0,0,0,0,0,0,0,0,0,0
P00034=-0.304,0.773,-2.693,0.0000,0.0000,0.0000
P00035=2.817,0.591,-1.622,0.0000,0.0000,0.0000
P00040=-0.030,9.648,2.467,0.0000,0.0000,0.0000
P00041=0.192,3.924,0.305,0.0000,0.0000,0.0000
P00042=-0.217,1.941,0.413,0.0000,0.0000,0.0000
P00043=-0.044,-1.937,1.197,0.0000,0.0000,0.0000
P00044=0.687,-2.322,1.156,0.0000,0.0000,0.0000
P00045=-0.068,-0.810,1.603,0.0000,0.0000,0.0000
P00046=0.799,0.043,1.292,0.0000,0.0000,0.0000
///RCONF 0,1,0,0,0,0,0,0,0,0,0,0,0,0,0,0,0,0,0,0,0,0,0,0
P00047=-0.011,1.737,-0.646,0.0000,0.0000,0.0000
///RCONF 0,0,0,0,0,0,0,0,0,0,0,0,0,0,0,0,0,0,0,0,0,0,0,0
P00048=2.411,0.025,-0.606,0.0000,0.0000,0.0000
P00049=3.413,-3.572,-1.618,0.0000,0.0000,0.0000
P00050=4.296,-4.501,-0.826,0.0000,0.0000,0.0000
P00051=0.367,3.892,0.009,0.0000,0.0000,0.0000
P00052=0.088,2.832,-0.342,0.0000,0.0000,0.0000
P00053=0.134,6.594,0.107,0.0000,0.0000,0.0000
P00054=-0.103,6.509,-0.702,0.0000,0.0000,0.0000
P00061=1.575,-3.405,-0.752,0.0000,0.0000,0.0000
P00062=-0.135,-0.848,-1.706,0.0000,0.0000,0.0000
P00063=0.036,-0.654,-3.005,0.0000,0.0000,0.0000
P00071=2.716,0.070,1.352,0.0000,0.0000,0.0000
P00072=1.041,-0.003,-0.797,0.0000,0.0000,0.0000
P00073=-0.961,5.319,-6.157,0.0000,0.0000,0.0000
P00074=1.123,1.944,-5.914,0.0000,0.0000,0.0000
P00088=-2.376,0.094,2.453,0.0000,0.0000,0.0000
P00089=5.697,-3.100,-1.263,0.0000,0.0000,0.0000
P00095=-3.945,4.918,-0.177,0.0000,0.0000,0.0000
P00096=-0.633,5.398,-3.809,0.0000,0.0000,0.0000
//INST
///DATE 2024/11/04 13:45
///ATTR SC,RW
///GROUP1 RB1,BS1
///GROUP2 ST1
NOP
'X2_8B-21B(90,180)
'
MOVJ C00000 BC00000 VJ=100.00  +MOVJ EC00000 VJ=100.00
'Path S4722
SFTOF3D
MOVJ C00001 BC00001 VJ=100.00  +MOVJ EC00001 VJ=100.00
MOVL C00002 BC00002 V=666.7  +MOVJ EC00002 VJ=100.00
SMOVL C00003 BC00003 V=166.7  +MOVJ EC00003
SREFP 3 C00004 BC00004  +REFP EC00004
CALL JOB:SEARCH-R1-S13D
SET P095 P006
SFTON3D P095
SMOVL C00005 BC00005 V=166.7  +MOVJ EC00005
SREFP 3 C00006 BC00006  +REFP EC00006
CALL JOB:SEARCH-R1-S13D
SET P095 P006
SFTON3D P095
SMOVL C00007 BC00007 V=166.7  +MOVJ EC00007
MOVL C00008 BC00008 V=1000.0  +MOVJ EC00008 VJ=100.00
'EndPath S4722
'Path S4723
SFTOF3D
MOVJ C00009 BC00009 VJ=100.00  +MOVJ EC00009 VJ=100.00
MOVL C00010 BC00010 V=666.7  +MOVJ EC00010 VJ=100.00
SMOVL C00011 BC00011 V=166.7  +MOVJ EC00011
SREFP 3 C00012 BC00012  +REFP EC00012
CALL JOB:SEARCH-R1-S13D
SET P096 P006
SFTON3D P096
SMOVL C00013 BC00013 V=166.7  +MOVJ EC00013
SREFP 3 C00014 BC00014  +REFP EC00014
CALL JOB:SEARCH-R1-S13D
SET P096 P006
SFTON3D P096
SMOVL C00015 BC00015 V=166.7  +MOVJ EC00015
MOVL C00016 BC00016 V=1000.0  +MOVJ EC00016 VJ=100.00
'EndPath S4723
'
'
'Path S4093
SFTOF3D
MOVJ C00017 BC00017 VJ=100.00  +MOVJ EC00017 VJ=100.00
MOVL C00018 BC00018 V=666.7  +MOVJ EC00018 VJ=100.00
SMOVL C00019 BC00019 V=166.7  +MOVJ EC00019
SREFP 3 C00020 BC00020  +REFP EC00020
CALL JOB:SEARCH-R1-S13D
SET P021 P006
SFTON3D P021
SMOVL C00021 BC00021 V=166.7  +MOVJ EC00021
SREFP 3 C00022 BC00022  +REFP EC00022
CALL JOB:SEARCH-R1-S13D
SET P021 P006
SFTON3D P021
SMOVL C00023 BC00023 V=166.7  +MOVJ EC00023
MOVL C00024 BC00024 V=1000.0  +MOVJ EC00024 VJ=100.00
'EndPath S4093
'Path S4094
SFTOF3D
MOVJ C00025 BC00025 VJ=100.00  +MOVJ EC00025 VJ=100.00
MOVL C00026 BC00026 V=666.7  +MOVJ EC00026 VJ=100.00
SMOVL C00027 BC00027 V=166.7  +MOVJ EC00027
SREFP 3 C00028 BC00028  +REFP EC00028
CALL JOB:SEARCH-R1-S13D
SET P022 P006
SFTON3D P022
SMOVL C00029 BC00029 V=166.7  +MOVJ EC00029
SREFP 3 C00030 BC00030  +REFP EC00030
CALL JOB:SEARCH-R1-S13D
SET P022 P006
SFTON3D P022
SMOVL C00031 BC00031 V=166.7  +MOVJ EC00031
MOVL C00032 BC00032 V=1000.0  +MOVJ EC00032 VJ=100.00
'EndPath S4094
MOVJ C00033 BC00033 VJ=100.00  +MOVJ EC00033 VJ=100.00
'Path S4205
SFTOF3D
MOVJ C00034 BC00034 VJ=100.00  +MOVJ EC00034 VJ=100.00
MOVL C00035 BC00035 V=666.7  +MOVJ EC00035 VJ=100.00
SMOVL C00036 BC00036 V=166.7  +MOVJ EC00036
SREFP 3 C00037 BC00037  +REFP EC00037
CALL JOB:SEARCH-R1-S13D
SET P050 P006
SFTON3D P050
SMOVL C00038 BC00038 V=166.7  +MOVJ EC00038
SREFP 3 C00039 BC00039  +REFP EC00039
CALL JOB:SEARCH-R1-S13D
SET P050 P006
SFTON3D P050
SMOVL C00040 BC00040 V=166.7  +MOVJ EC00040
SMOVL C00041 BC00041 V=250.0  +MOVJ EC00041
SMOVL C00042 BC00042 V=166.7  +MOVJ EC00042
SREFP 3 C00043 BC00043  +REFP EC00043
CALL JOB:SEARCH-R1-S13D
SET P050 P006
SFTON3D P050
SMOVL C00044 BC00044 V=250.0  +MOVJ EC00044
'EndPath S4205
'Path S4206
SFTOF3D
MOVL C00045 BC00045 V=1000.0  +MOVJ EC00045 VJ=100.00
SMOVL C00046 BC00046 V=166.7  +MOVJ EC00046
SREFP 3 C00047 BC00047  +REFP EC00047
CALL JOB:SEARCH-R1-S13D
SET P051 P006
SFTON3D P051
SMOVL C00048 BC00048 V=166.7  +MOVJ EC00048
SREFP 3 C00049 BC00049  +REFP EC00049
CALL JOB:SEARCH-R1-S13D
SET P051 P006
SFTON3D P051
SMOVL C00050 BC00050 V=166.7  +MOVJ EC00050
SMOVL C00051 BC00051 V=250.0  +MOVJ EC00051
SREFP 3 C00052 BC00052  +REFP EC00052
CALL JOB:SEARCH-R1-S13D
SET P051 P006
SFTON3D P051
SMOVL C00053 BC00053 V=250.0  +MOVJ EC00053
MOVL C00054 BC00054 V=1000.0  +MOVJ EC00054 VJ=100.00
'EndPath S4206
MOVJ C00055 BC00055 VJ=100.00  +MOVJ EC00055 VJ=100.00
'Path S4207
SFTOF3D
MOVJ C00056 BC00056 VJ=100.00  +MOVJ EC00056 VJ=100.00
MOVL C00057 BC00057 V=666.7  +MOVJ EC00057 VJ=100.00
SMOVL C00058 BC00058 V=166.7  +MOVJ EC00058
SREFP 3 C00059 BC00059  +REFP EC00059
CALL JOB:SEARCH-R1-S13D
SET P054 P006
SFTON3D P054
SMOVL C00060 BC00060 V=250.0  +MOVJ EC00060
SMOVL C00061 BC00061 V=233.3  +MOVJ EC00061
SMOVL C00062 BC00062 V=166.7  +MOVJ EC00062
